C03641=1077.730,297.238,-89.064,175.217,27.521,154.780
C03642=1077.736,297.486,-89.094,175.220,27.526,154.780
C03643=1077.741,297.734,-89.125,175.222,27.530,154.781
C03644=1077.748,297.982,-89.156,175.225,27.534,154.781
C03645=1077.753,298.230,-89.187,175.228,27.538,154.782
C03646=1077.759,298.478,-89.218,175.231,27.542,154.783
C03647=1077.764,298.725,-89.249,175.234,27.547,154.783
C03648=1077.771,298.974,-89.280,175.236,27.551,154.784
C03649=1077.776,299.221,-89.312,175.240,27.555,154.785
C03650=1077.782,299.469,-89.342,175.242,27.559,154.785
C03651=1077.788,299.718,-89.373,175.245,27.563,154.786
C03652=1077.794,299.965,-89.404,175.248,27.567,154.787
C03653=1077.799,300.213,-89.435,175.251,27.571,154.787
C03654=1077.805,300.462,-89.467,175.254,27.576,154.788
C03655=1077.811,300.709,-89.498,175.257,27.580,154.789
C03656=1077.816,300.957,-89.529,175.259,27.584,154.789
C03657=1077.823,301.205,-89.561,175.262,27.588,154.790
C03658=1077.828,301.453,-89.592,175.265,27.592,154.791
C03659=1077.834,301.701,-89.624,175.268,27.596,154.791
C03660=1077.840,301.949,-89.654,175.271,27.601,154.792
C03661=1077.845,302.197,-89.686,175.273,27.605,154.793
C03662=1077.851,302.445,-89.717,175.277,27.609,154.793
C03663=1077.857,302.693,-89.748,175.280,27.614,154.794
C03664=1077.863,302.916,-89.777,175.282,27.617,154.794
C03665=1077.867,303.139,-89.805,175.284,27.621,154.795
C03666=1077.873,303.363,-89.833,175.288,27.625,154.796
C03667=1077.878,303.586,-89.862,175.290,27.629,154.796
C03668=1077.883,303.809,-89.890,175.292,27.632,154.797
C03669=1077.888,304.032,-89.919,175.295,27.636,154.797
C03670=1077.894,304.256,-89.946,175.298,27.640,154.798
C03671=1077.899,304.479,-89.975,175.300,27.644,154.799
C03672=1077.905,304.716,-90.005,175.303,27.647,154.799
C03673=1077.911,304.953,-90.034,175.306,27.651,154.800
C03674=1077.916,305.190,-90.065,175.309,27.656,154.800
C03675=1077.922,305.426,-90.096,175.311,27.660,154.801
C03676=1077.927,305.663,-90.125,175.314,27.664,154.802
C03677=1077.932,305.900,-90.155,175.317,27.667,154.802
C03678=1077.938,306.136,-90.185,175.320,27.672,154.803
C03679=1077.944,306.374,-90.216,175.322,27.676,154.804
C03680=1077.950,306.621,-90.247,175.326,27.680,154.804
C03681=1077.956,306.870,-90.279,175.329,27.684,154.805
C03682=1077.961,307.117,-90.310,175.331,27.689,154.806
C03683=1077.967,307.365,-90.342,175.334,27.693,154.806
C03684=1077.974,307.613,-90.373,175.337,27.697,154.807
C03685=1077.980,307.861,-90.405,175.340,27.701,154.808
C03686=1077.986,308.109,-90.438,175.343,27.705,154.808
C03687=1077.992,308.356,-90.469,175.346,27.709,154.809
C03688=1077.998,308.604,-90.501,175.349,27.714,154.810
C03689=1078.003,308.852,-90.532,175.352,27.718,154.810
C03690=1078.009,309.100,-90.564,175.355,27.722,154.811
C03691=1078.016,309.348,-90.596,175.358,27.727,154.812
C03692=1078.021,309.596,-90.627,175.360,27.731,154.812
C03693=1078.027,309.844,-90.659,175.364,27.735,154.813
C03694=1078.033,310.092,-90.691,175.367,27.739,154.814
C03695=1078.039,310.339,-90.722,175.370,27.743,154.814
C03696=1078.046,310.587,-90.755,175.372,27.748,154.815
C03697=1078.052,310.835,-90.787,175.376,27.752,154.816
C03698=1078.058,311.083,-90.819,175.379,27.756,154.816
C03699=1078.063,311.331,-90.851,175.381,27.760,154.817
C03700=1078.070,311.579,-90.882,175.384,27.764,154.818
C03701=1078.076,311.827,-90.914,175.387,27.769,154.818
C03702=1078.082,312.074,-90.947,175.391,27.773,154.819
C03703=1078.087,312.322,-90.979,175.393,27.777,154.820
C03704=1078.093,312.570,-91.011,175.396,27.782,154.820
C03705=1078.100,312.818,-91.042,175.399,27.786,154.821
C03706=1078.106,313.066,-91.075,175.403,27.791,154.822
C03707=1078.112,313.313,-91.107,175.405,27.794,154.822
C03708=1078.118,313.561,-91.139,175.408,27.799,154.823
C03709=1078.124,313.810,-91.171,175.411,27.803,154.824
C03710=1078.130,314.057,-91.203,175.415,27.808,154.824
C03711=1078.137,314.305,-91.235,175.417,27.812,154.825
C03712=1078.143,314.553,-91.267,175.420,27.816,154.826
C03713=1078.148,314.800,-91.299,175.423,27.820,154.826
C03714=1078.154,315.049,-91.332,175.427,27.825,154.827
C03715=1078.160,315.296,-91.365,175.429,27.829,154.828
C03716=1078.166,315.545,-91.397,175.432,27.833,154.829
C03717=1078.172,315.791,-91.429,175.435,27.838,154.829
C03718=1078.177,316.040,-91.462,175.438,27.842,154.830
C03719=1078.183,316.288,-91.494,175.441,27.847,154.831
C03720=1078.188,316.501,-91.522,175.444,27.851,154.831
C03721=1078.193,316.716,-91.550,175.446,27.855,154.832
C03722=1078.198,316.929,-91.578,175.449,27.858,154.833
C03723=1078.202,317.143,-91.606,175.451,27.862,154.833
C03724=1078.208,317.356,-91.634,175.454,27.866,154.834
C03725=1078.212,317.570,-91.662,175.456,27.870,154.835
C03726=1078.218,317.784,-91.690,175.459,27.874,154.835
C03727=1078.223,317.998,-91.718,175.461,27.878,154.836
C03728=1078.229,318.245,-91.751,175.464,27.882,154.836
C03729=1078.235,318.493,-91.784,175.468,27.887,154.837
C03730=1078.240,318.742,-91.816,175.471,27.892,154.838
C03731=1078.247,318.989,-91.849,175.474,27.896,154.839
C03732=1078.253,319.237,-91.882,175.476,27.900,154.839
C03733=1078.258,319.485,-91.914,175.479,27.905,154.840
C03734=1078.264,319.732,-91.947,175.483,27.909,154.841
C03735=1078.270,319.980,-91.980,175.486,27.914,154.842
C03736=1078.276,320.228,-92.013,175.489,27.919,154.842
C03737=1078.282,320.476,-92.045,175.491,27.923,154.843
C03738=1078.288,320.723,-92.078,175.494,27.927,154.844
C03739=1078.294,320.971,-92.111,175.498,27.932,154.845
C03740=1078.300,321.219,-92.144,175.501,27.936,154.845
C03741=1078.305,321.467,-92.177,175.504,27.941,154.846
C03742=1078.311,321.715,-92.209,175.506,27.945,154.847
C03743=1078.318,321.963,-92.242,175.509,27.950,154.848
C03744=1078.323,322.210,-92.275,175.513,27.954,154.848
C03745=1078.329,322.457,-92.308,175.516,27.959,154.849
C03746=1078.335,322.705,-92.340,175.519,27.964,154.850
C03747=1078.341,322.953,-92.374,175.522,27.968,154.851
C03748=1078.347,323.201,-92.406,175.525,27.972,154.851
C03749=1078.353,323.448,-92.440,175.528,27.977,154.852
C03750=1078.359,323.696,-92.472,175.531,27.982,154.853
C03751=1078.364,323.944,-92.506,175.534,27.987,154.854
C03752=1078.371,324.192,-92.539,175.537,27.991,154.854
C03753=1078.378,324.440,-92.572,175.541,27.995,154.855
C03754=1078.383,324.688,-92.605,175.544,28.000,154.856
C03755=1078.390,324.935,-92.638,175.546,28.005,154.857
C03756=1078.395,325.183,-92.671,175.549,28.009,154.857
C03757=1078.401,325.431,-92.704,175.552,28.014,154.858
C03758=1078.407,325.679,-92.737,175.556,28.018,154.859
C03759=1078.413,325.926,-92.770,175.559,28.023,154.859
C03760=1078.419,326.174,-92.803,175.562,28.028,154.860
C03761=1078.425,326.422,-92.836,175.565,28.032,154.861
C03762=1078.431,326.669,-92.870,175.568,28.037,154.862
C03763=1078.437,326.917,-92.903,175.571,28.041,154.863
C03764=1078.443,327.165,-92.936,175.574,28.046,154.863
C03765=1078.450,327.413,-92.969,175.577,28.050,154.864
C03766=1078.455,327.661,-93.003,175.580,28.055,154.865
C03767=1078.462,327.908,-93.036,175.584,28.060,154.866
C03768=1078.467,328.156,-93.069,175.587,28.064,154.866
C03769=1078.474,328.403,-93.102,175.590,28.069,154.867
C03770=1078.480,328.652,-93.136,175.593,28.074,154.868
C03771=1078.486,328.899,-93.169,175.596,28.078,154.869
C03772=1078.492,329.147,-93.203,175.599,28.083,154.869
C03773=1078.498,329.394,-93.235,175.602,28.088,154.870
C03774=1078.504,329.642,-93.269,175.605,28.092,154.871
C03775=1078.511,329.890,-93.303,175.608,28.097,154.872
C03776=1078.516,330.100,-93.331,175.612,28.101,154.872
C03777=1078.522,330.311,-93.360,175.614,28.105,154.873
C03778=1078.526,330.521,-93.388,175.616,28.108,154.874
C03779=1078.531,330.732,-93.416,175.620,28.113,154.874
C03780=1078.537,330.943,-93.445,175.622,28.117,154.875
C03781=1078.541,331.153,-93.473,175.624,28.120,154.876
C03782=1078.547,331.364,-93.502,175.628,28.125,154.876
C03783=1078.552,331.574,-93.531,175.630,28.129,154.877
C03784=1078.559,331.821,-93.564,175.633,28.134,154.878
C03785=1078.564,332.069,-93.597,175.636,28.138,154.879
C03786=1078.571,332.317,-93.632,175.639,28.143,154.879
C03787=1078.576,332.565,-93.665,175.643,28.148,154.880
C03788=1078.582,332.812,-93.699,175.646,28.153,154.881
C03789=1078.588,333.059,-93.733,175.649,28.158,154.882
C03790=1078.594,333.308,-93.767,175.651,28.162,154.883
C03791=1078.600,333.555,-93.801,175.654,28.167,154.884
C03792=1078.606,333.803,-93.834,175.658,28.172,154.884
C03793=1078.612,334.050,-93.868,175.661,28.177,154.885
C03794=1078.619,334.298,-93.902,175.664,28.182,154.886
C03795=1078.625,334.546,-93.936,175.667,28.186,154.887
C03796=1078.630,334.793,-93.970,175.670,28.191,154.888
C03797=1078.637,335.041,-94.004,175.674,28.196,154.888
C03798=1078.642,335.289,-94.038,175.677,28.201,154.889
C03799=1078.648,335.536,-94.072,175.680,28.206,154.890
C03800=1078.654,335.785,-94.106,175.683,28.211,154.891
C03801=1078.660,336.032,-94.140,175.686,28.216,154.892
C03802=1078.666,336.279,-94.174,175.689,28.221,154.893
C03803=1078.673,336.527,-94.208,175.693,28.225,154.893
C03804=1078.678,336.774,-94.242,175.696,28.230,154.894
C03805=1078.685,337.021,-94.276,175.699,28.235,154.895
C03806=1078.691,337.270,-94.310,175.702,28.240,154.896
C03807=1078.697,337.517,-94.344,175.705,28.245,154.897
C03808=1078.704,337.765,-94.378,175.709,28.250,154.897
C03809=1078.709,338.013,-94.412,175.712,28.255,154.898
C03810=1078.715,338.260,-94.447,175.715,28.260,154.899
C03811=1078.721,338.508,-94.481,175.718,28.265,154.900
C03812=1078.727,338.755,-94.515,175.721,28.270,154.901
C03813=1078.733,339.003,-94.550,175.725,28.275,154.902
C03814=1078.739,339.251,-94.584,175.728,28.280,154.903
C03815=1078.745,339.498,-94.618,175.731,28.285,154.904
C03816=1078.752,339.745,-94.653,175.734,28.290,154.904
C03817=1078.757,339.993,-94.687,175.737,28.295,154.905
C03818=1078.763,340.241,-94.722,175.740,28.300,154.906
C03819=1078.769,340.488,-94.756,175.744,28.305,154.907
C03820=1078.776,340.736,-94.790,175.747,28.310,154.908
C03821=1078.782,340.983,-94.824,175.750,28.315,154.909
C03822=1078.788,341.231,-94.859,175.753,28.320,154.910
C03823=1078.793,341.478,-94.894,175.757,28.326,154.910
C03824=1078.799,341.726,-94.928,175.760,28.330,154.911
C03825=1078.806,341.974,-94.963,175.764,28.335,154.912
C03826=1078.812,342.222,-94.997,175.767,28.341,154.913
C03827=1078.818,342.468,-95.032,175.770,28.346,154.914
C03828=1078.824,342.717,-95.067,175.773,28.351,154.915
C03829=1078.830,342.964,-95.101,175.776,28.356,154.916
C03830=1078.837,343.211,-95.136,175.780,28.361,154.917
C03831=1078.843,343.459,-95.170,175.783,28.366,154.917
C03832=1078.853,343.875,-95.229,175.788,28.374,154.919
C03833=1078.863,344.290,-95.287,175.794,28.383,154.920
C03834=1078.873,344.706,-95.345,175.800,28.392,154.922
C03835=1078.883,345.122,-95.404,175.804,28.400,154.923
C03836=1078.890,345.369,-95.439,175.808,28.406,154.924
C03837=1078.895,345.617,-95.474,175.811,28.411,154.925
C03838=1078.902,345.863,-95.508,175.815,28.416,154.926
C03839=1078.907,346.112,-95.543,175.818,28.422,154.927
C03840=1078.914,346.359,-95.578,175.821,28.427,154.928
C03841=1078.920,346.606,-95.613,175.824,28.432,154.929
C03842=1078.926,346.854,-95.648,175.827,28.437,154.930
C03843=1078.932,347.101,-95.683,175.830,28.442,154.931
C03844=1078.938,347.349,-95.718,175.834,28.448,154.932
C03845=1078.945,347.596,-95.753,175.838,28.453,154.933
C03846=1078.950,347.843,-95.789,175.841,28.458,154.934
C03847=1078.956,348.091,-95.823,175.844,28.463,154.934
C03848=1078.962,348.339,-95.859,175.847,28.469,154.935
C03849=1078.969,348.586,-95.893,175.850,28.474,154.936
C03850=1078.975,348.833,-95.929,175.854,28.479,154.937
C03851=1078.981,349.081,-95.964,175.857,28.485,154.938
C03852=1078.987,349.328,-95.999,175.861,28.490,154.939
C03853=1078.993,349.576,-96.035,175.864,28.496,154.940
C03854=1078.999,349.823,-96.070,175.867,28.501,154.941
C03855=1079.005,350.070,-96.105,175.870,28.506,154.942
C03856=1079.012,350.318,-96.140,175.874,28.512,154.943
C03857=1079.017,350.566,-96.175,175.877,28.517,154.944
C03858=1079.024,350.813,-96.210,175.880,28.522,154.945
C03859=1079.029,351.060,-96.246,175.884,28.528,154.946
C03860=1079.036,351.308,-96.282,175.887,28.533,154.947
C03861=1079.042,351.555,-96.317,175.890,28.538,154.948
C03862=1079.048,351.803,-96.352,175.893,28.544,154.949
C03863=1079.054,352.050,-96.388,175.897,28.549,154.950
C03864=1079.061,352.297,-96.423,175.901,28.555,154.951
C03865=1079.067,352.545,-96.459,175.904,28.560,154.952
C03866=1079.073,352.793,-96.494,175.907,28.566,154.953
C03867=1079.079,353.039,-96.529,175.910,28.571,154.954
C03868=1079.085,353.287,-96.565,175.913,28.577,154.955
C03869=1079.091,353.534,-96.601,175.917,28.583,154.956
C03870=1079.097,353.782,-96.637,175.921,28.588,154.956
C03871=1079.104,354.029,-96.672,175.924,28.593,154.957
C03872=1079.109,354.276,-96.708,175.927,28.599,154.959
C03873=1079.115,354.524,-96.743,175.930,28.605,154.960
C03874=1079.121,354.772,-96.779,175.934,28.610,154.960
C03875=1079.128,355.019,-96.815,175.937,28.616,154.961
C03876=1079.134,355.266,-96.851,175.941,28.621,154.962
C03877=1079.141,355.514,-96.886,175.944,28.627,154.964
C03878=1079.146,355.761,-96.922,175.947,28.632,154.965
C03879=1079.152,356.008,-96.958,175.951,28.638,154.966
C03880=1079.158,356.255,-96.994,175.954,28.643,154.966
C03881=1079.164,356.503,-97.030,175.957,28.649,154.968
C03882=1079.171,356.750,-97.066,175.960,28.655,154.969
C03883=1079.177,356.997,-97.101,175.965,28.660,154.970
C03884=1079.182,357.207,-97.132,175.967,28.665,154.970
C03885=1079.188,357.417,-97.162,175.970,28.670,154.971
C03886=1079.193,357.626,-97.192,175.972,28.675,154.972
C03887=1079.198,357.835,-97.223,175.976,28.679,154.973
C03888=1079.204,358.045,-97.254,175.979,28.684,154.974
C03889=1079.208,358.254,-97.284,175.981,28.689,154.975
C03890=1079.214,358.463,-97.314,175.984,28.694,154.976
C03891=1079.219,358.673,-97.345,175.988,28.699,154.977
C03892=1079.226,358.920,-97.381,175.991,28.705,154.978
C03893=1079.232,359.168,-97.417,175.994,28.710,154.979
C03894=1079.238,359.415,-97.454,175.997,28.716,154.980
C03895=1079.244,359.662,-97.489,176.001,28.722,154.981
C03896=1079.250,359.909,-97.526,176.004,28.728,154.982
C03897=1079.257,360.156,-97.562,176.008,28.733,154.983
C03898=1079.263,360.404,-97.598,176.012,28.739,154.984
C03899=1079.269,360.651,-97.634,176.015,28.745,154.985
C03900=1079.276,360.898,-97.671,176.018,28.751,154.986
C03901=1079.282,361.145,-97.707,176.021,28.757,154.987
C03902=1079.288,361.393,-97.743,176.025,28.762,154.988
C03903=1079.293,361.640,-97.780,176.028,28.769,154.989
C03904=1079.300,361.887,-97.816,176.031,28.774,154.990
C03905=1079.306,362.134,-97.853,176.036,28.780,154.991
C03906=1079.312,362.382,-97.889,176.039,28.786,154.992
C03907=1079.319,362.629,-97.925,176.042,28.792,154.993
C03908=1079.325,362.876,-97.962,176.046,28.798,154.995
C03909=1079.331,363.123,-97.998,176.049,28.804,154.996
C03910=1079.338,363.370,-98.034,176.052,28.810,154.997
C03911=1079.343,363.618,-98.071,176.056,28.816,154.998
C03912=1079.349,363.865,-98.108,176.059,28.822,154.999
C03913=1079.356,364.112,-98.144,176.063,28.827,155.000
C03914=1079.362,364.359,-98.181,176.067,28.834,155.001
C03915=1079.369,364.607,-98.218,176.070,28.839,155.002
C03916=1079.375,364.854,-98.255,176.073,28.845,155.003
C03917=1079.381,365.101,-98.291,176.077,28.852,155.005
C03918=1079.387,365.348,-98.328,176.080,28.857,155.006
C03919=1079.394,365.595,-98.364,176.083,28.863,155.007
C03920=1079.399,365.842,-98.401,176.087,28.870,155.008
C03921=1079.406,366.090,-98.437,176.091,28.876,155.009
C03922=1079.411,366.337,-98.475,176.095,28.882,155.010
C03923=1079.418,366.585,-98.511,176.098,28.888,155.011
C03924=1079.425,366.831,-98.549,176.101,28.894,155.012
C03925=1079.430,367.078,-98.586,176.105,28.900,155.014
C03926=1079.437,367.325,-98.622,176.108,28.906,155.015
C03927=1079.442,367.573,-98.659,176.111,28.912,155.016
C03928=1079.449,367.819,-98.696,176.115,28.918,155.017
C03929=1079.456,368.067,-98.733,176.119,28.925,155.018
C03930=1079.462,368.314,-98.770,176.123,28.931,155.019
C03931=1079.468,368.561,-98.806,176.126,28.937,155.021
C03932=1079.474,368.808,-98.844,176.129,28.944,155.022
C03933=1079.480,369.055,-98.881,176.133,28.950,155.023
C03934=1079.487,369.303,-98.919,176.136,28.956,155.024
C03935=1079.493,369.550,-98.955,176.140,28.962,155.025
C03936=1079.499,369.797,-98.992,176.143,28.968,155.026
C03937=1079.505,370.044,-99.029,176.146,28.974,155.028
C03938=1079.512,370.291,-99.066,176.150,28.981,155.029
C03939=1079.518,370.538,-99.104,176.154,28.987,155.030
C03940=1079.524,370.755,-99.137,176.157,28.993,155.031
C03941=1079.529,370.973,-99.169,176.160,28.998,155.032
C03942=1079.535,371.190,-99.202,176.163,29.004,155.033
C03943=1079.541,371.408,-99.235,176.166,29.009,155.034
C03944=1079.546,371.626,-99.268,176.170,29.015,155.035
C03945=1079.552,371.843,-99.300,176.173,29.021,155.036
C03946=1079.557,372.060,-99.333,176.176,29.026,155.037
C03947=1079.563,372.278,-99.367,176.179,29.032,155.038
C03948=1079.569,372.525,-99.404,176.182,29.038,155.040
C03949=1079.576,372.772,-99.441,176.187,29.045,155.041
C03950=1079.582,373.019,-99.479,176.190,29.051,155.042
C03951=1079.588,373.267,-99.516,176.194,29.057,155.043
C03952=1079.595,373.514,-99.554,176.197,29.064,155.044
C03953=1079.601,373.761,-99.591,176.201,29.070,155.046
C03954=1079.608,374.007,-99.628,176.204,29.077,155.047
C03955=1079.614,374.255,-99.666,176.208,29.084,155.048
C03956=1079.620,374.502,-99.704,176.211,29.090,155.049
C03957=1079.626,374.749,-99.741,176.214,29.096,155.051
C03958=1079.632,374.996,-99.779,176.218,29.103,155.052
C03959=1079.639,375.242,-99.817,176.222,29.109,155.053
C03960=1079.645,375.489,-99.854,176.226,29.116,155.054
C03961=1079.651,375.737,-99.892,176.229,29.123,155.056
C03962=1079.657,375.983,-99.930,176.233,29.130,155.057
C03963=1079.664,376.231,-99.968,176.237,29.136,155.058
C03964=1079.670,376.477,-100.006,176.240,29.143,155.060
C03965=1079.677,376.725,-100.044,176.244,29.150,155.061
C03966=1079.683,376.971,-100.081,176.247,29.156,155.062
C03967=1079.689,377.219,-100.120,176.251,29.163,155.063
C03968=1079.695,377.466,-100.157,176.254,29.170,155.065
C03969=1079.702,377.713,-100.195,176.259,29.176,155.066
C03970=1079.708,377.959,-100.233,176.262,29.183,155.067
C03971=1079.715,378.207,-100.271,176.266,29.190,155.069
C03972=1079.721,378.453,-100.309,176.269,29.197,155.070
C03973=1079.727,378.701,-100.347,176.273,29.203,155.071
C03974=1079.733,378.947,-100.385,176.276,29.210,155.073
C03975=1079.740,379.195,-100.423,176.280,29.217,155.074
C03976=1079.746,379.441,-100.462,176.284,29.224,155.075
C03977=1079.753,379.688,-100.499,176.287,29.231,155.076
C03978=1079.759,379.935,-100.537,176.291,29.237,155.078
C03979=1079.766,380.182,-100.576,176.294,29.244,155.079
C03980=1079.773,380.429,-100.614,176.299,29.251,155.080
C03981=1079.778,380.676,-100.652,176.303,29.258,155.082
C03982=1079.785,380.923,-100.690,176.306,29.265,155.083
C03983=1079.791,381.169,-100.728,176.310,29.272,155.084
C03984=1079.798,381.416,-100.767,176.313,29.279,155.086
C03985=1079.804,381.664,-100.805,176.317,29.285,155.087
C03986=1079.811,381.911,-100.843,176.321,29.293,155.089
C03987=1079.817,382.157,-100.882,176.324,29.300,155.090
C03988=1079.824,382.405,-100.920,176.328,29.306,155.091
C03989=1079.830,382.651,-100.958,176.332,29.314,155.093
C03990=1079.837,382.897,-100.997,176.335,29.321,155.094
C03991=1079.843,383.145,-101.035,176.339,29.328,155.095
C03992=1079.849,383.391,-101.074,176.343,29.335,155.097
C03993=1079.855,383.638,-101.113,176.347,29.342,155.098
C03994=1079.862,383.886,-101.151,176.351,29.349,155.100
C03995=1079.868,384.132,-101.190,176.354,29.356,155.101
C03996=1079.874,384.364,-101.226,176.358,29.363,155.102
C03997=1079.880,384.595,-101.263,176.361,29.370,155.104
C03998=1079.886,384.827,-101.299,176.364,29.377,155.105
C03999=1079.892,385.059,-101.336,176.368,29.383,155.106
C04000=1079.898,385.291,-101.372,176.371,29.390,155.108
C04001=1079.905,385.523,-101.408,176.376,29.397,155.109
C04002=1079.910,385.755,-101.445,176.379,29.404,155.110
C04003=1079.917,385.987,-101.481,176.382,29.411,155.112
C04004=1079.923,386.234,-101.520,176.386,29.418,155.113
C04005=1079.929,386.480,-101.559,176.390,29.425,155.115
C04006=1079.936,386.727,-101.597,176.394,29.433,155.116
C04007=1079.943,386.974,-101.636,176.397,29.440,155.118
C04008=1079.949,387.221,-101.676,176.401,29.447,155.119
C04009=1079.955,387.467,-101.714,176.405,29.455,155.120
C04010=1079.962,387.714,-101.753,176.408,29.462,155.122
C04011=1079.968,387.961,-101.792,176.413,29.469,155.123
C04012=1079.974,388.208,-101.831,176.417,29.477,155.125
C04013=1079.981,388.455,-101.870,176.421,29.484,155.126
C04014=1079.988,388.701,-101.909,176.424,29.492,155.128
C04015=1079.994,388.949,-101.948,176.428,29.499,155.129
C04016=1080.001,389.194,-101.988,176.432,29.507,155.131
C04017=1080.008,389.441,-102.026,176.436,29.514,155.132
C04018=1080.014,389.688,-102.066,176.439,29.521,155.134
C04019=1080.020,389.935,-102.105,176.443,29.529,155.135
C04020=1080.027,390.182,-102.144,176.447,29.537,155.137
C04021=1080.034,390.428,-102.184,176.451,29.544,155.138
C04022=1080.040,390.675,-102.223,176.455,29.552,155.140
C04023=1080.047,390.922,-102.261,176.458,29.559,155.141
C04024=1080.054,391.168,-102.302,176.463,29.567,155.143
C04025=1080.060,391.415,-102.340,176.467,29.574,155.144
C04026=1080.066,391.662,-102.380,176.471,29.582,155.146
C04027=1080.074,391.908,-102.419,176.475,29.590,155.147
C04028=1080.080,392.156,-102.459,176.478,29.597,155.149
C04029=1080.087,392.402,-102.498,176.482,29.606,155.151
C04030=1080.093,392.649,-102.538,176.486,29.613,155.152
C04031=1080.099,392.895,-102.578,176.490,29.621,155.154
C04032=1080.106,393.142,-102.617,176.494,29.629,155.155
C04033=1080.112,393.389,-102.657,176.497,29.636,155.157
C04034=1080.119,393.636,-102.696,176.501,29.644,155.158
C04035=1080.126,393.882,-102.736,176.505,29.652,155.160
C04036=1080.132,394.129,-102.776,176.509,29.660,155.162
C04037=1080.139,394.375,-102.815,176.513,29.668,155.163
C04038=1080.145,394.622,-102.855,176.518,29.676,155.165
C04039=1080.152,394.869,-102.896,176.521,29.684,155.167
C04040=1080.159,395.116,-102.934,176.525,29.692,155.168
C04041=1080.165,395.363,-102.975,176.529,29.700,155.170
C04042=1080.172,395.609,-103.015,176.533,29.708,155.171
C04043=1080.178,395.856,-103.055,176.537,29.716,155.173
C04044=1080.185,396.102,-103.094,176.541,29.724,155.175
C04045=1080.191,396.349,-103.134,176.545,29.732,155.176
C04046=1080.198,396.596,-103.174,176.548,29.740,155.178
C04047=1080.205,396.843,-103.214,176.552,29.748,155.180
C04048=1080.211,397.089,-103.255,176.556,29.756,155.181
C04049=1080.218,397.335,-103.294,176.560,29.765,155.183
C04050=1080.225,397.582,-103.334,176.564,29.773,155.185
C04051=1080.232,397.829,-103.375,176.568,29.781,155.186
C04052=1080.238,398.068,-103.414,176.572,29.789,155.188
C04053=1080.244,398.307,-103.452,176.577,29.797,155.190
C04054=1080.250,398.546,-103.491,176.580,29.805,155.191
C04055=1080.258,398.785,-103.530,176.584,29.813,155.193
C04056=1080.264,399.024,-103.569,176.588,29.821,155.195
C04057=1080.270,399.263,-103.608,176.592,29.829,155.196
C04058=1080.276,399.502,-103.647,176.595,29.837,155.198
C04059=1080.283,399.741,-103.686,176.599,29.845,155.200
C04060=1080.289,399.988,-103.727,176.603,29.854,155.201
C04061=1080.296,400.234,-103.767,176.607,29.862,155.203
C04062=1080.303,400.481,-103.808,176.611,29.870,155.205
C04063=1080.309,400.727,-103.848,176.615,29.879,155.207
C04064=1080.316,400.974,-103.888,176.620,29.887,155.208
C04065=1080.323,401.221,-103.929,176.624,29.896,155.210
C04066=1080.329,401.467,-103.970,176.628,29.904,155.212
C04067=1080.336,401.714,-104.011,176.632,29.913,155.214
C04068=1080.342,401.961,-104.051,176.636,29.922,155.215
C04069=1080.349,402.207,-104.092,176.640,29.930,155.217
C04070=1080.356,402.454,-104.132,176.644,29.939,155.219
C04071=1080.363,402.700,-104.173,176.648,29.947,155.221
C04072=1080.370,402.947,-104.214,176.652,29.956,155.223
C04073=1080.376,403.193,-104.255,176.656,29.965,155.224
C04074=1080.383,403.440,-104.295,176.660,29.973,155.226
C04075=1080.390,403.686,-104.336,176.664,29.982,155.228
C04076=1080.397,403.933,-104.376,176.668,29.991,155.230
C04077=1080.403,404.180,-104.418,176.672,30.000,155.232
C04078=1080.410,404.426,-104.459,176.677,30.009,155.234
C04079=1080.416,404.673,-104.499,176.682,30.017,155.235
C04080=1080.424,404.919,-104.540,176.686,30.027,155.237
C04081=1080.430,405.165,-104.582,176.690,30.035,155.239
C04082=1080.437,405.413,-104.622,176.694,30.044,155.241
C04083=1080.443,405.659,-104.663,176.698,30.053,155.243
C04084=1080.451,405.905,-104.705,176.702,30.062,155.245
C04085=1080.457,406.152,-104.746,176.706,30.071,155.247
C04086=1080.464,406.398,-104.787,176.710,30.080,155.249
C04087=1080.471,406.645,-104.828,176.715,30.089,155.250
C04088=1080.477,406.891,-104.869,176.719,30.098,155.252
C04089=1080.484,407.138,-104.910,176.723,30.107,155.254
C04090=1080.491,407.385,-104.952,176.727,30.116,155.256
C04091=1080.497,407.631,-104.993,176.731,30.126,155.258
C04092=1080.504,407.878,-105.035,176.736,30.135,155.260
C04093=1080.511,408.124,-105.076,176.741,30.144,155.262
C04094=1080.517,408.370,-105.118,176.745,30.153,155.264
C04095=1080.524,408.617,-105.159,176.749,30.162,155.266
C04096=1080.530,408.863,-105.200,176.753,30.172,155.268
C04097=1080.538,409.109,-105.242,176.757,30.181,155.270
C04098=1080.544,409.356,-105.284,176.762,30.191,155.272
C04099=1080.551,409.602,-105.325,176.766,30.200,155.274
C04100=1080.558,409.849,-105.367,176.770,30.209,155.276
C04101=1080.565,410.096,-105.408,176.774,30.219,155.278
C04102=1080.572,410.342,-105.451,176.779,30.228,155.280
C04103=1080.579,410.588,-105.491,176.783,30.238,155.282
C04104=1080.585,410.835,-105.533,176.787,30.247,155.284
C04105=1080.593,411.081,-105.575,176.792,30.257,155.286
C04106=1080.599,411.328,-105.617,176.797,30.267,155.288
C04107=1080.606,411.574,-105.659,176.801,30.276,155.290
C04108=1080.612,411.814,-105.700,176.805,30.285,155.292
C04109=1080.619,412.054,-105.741,176.809,30.295,155.294
C04110=1080.626,412.294,-105.781,176.813,30.304,155.296
C04111=1080.633,412.534,-105.822,176.818,30.314,155.298
C04112=1080.640,412.774,-105.862,176.822,30.323,155.300
C04113=1080.647,413.014,-105.903,176.826,30.332,155.302
C04114=1080.653,413.255,-105.945,176.830,30.342,155.304
C04115=1080.660,413.494,-105.986,176.836,30.352,155.306
C04116=1080.667,413.741,-106.027,176.840,30.362,155.308
C04117=1080.674,413.987,-106.070,176.844,30.371,155.310
C04118=1080.681,414.234,-106.112,176.849,30.381,155.313
C04119=1080.688,414.480,-106.154,176.853,30.391,155.315
C04120=1080.695,414.727,-106.196,176.857,30.401,155.317
C04121=1080.702,414.973,-106.239,176.862,30.411,155.319
C04122=1080.709,415.219,-106.281,176.866,30.420,155.321
C04123=1080.716,415.466,-106.323,176.871,30.431,155.323
C04124=1080.723,415.712,-106.365,176.875,30.441,155.325
C04125=1080.730,415.958,-106.408,176.881,30.451,155.327
C04126=1080.737,416.205,-106.450,176.885,30.461,155.330
C04127=1080.743,416.451,-106.493,176.890,30.471,155.332
C04128=1080.751,416.697,-106.535,176.894,30.481,155.334
C04129=1080.758,416.943,-106.577,176.898,30.491,155.336
C04130=1080.765,417.189,-106.620,176.903,30.502,155.339
C04131=1080.772,417.436,-106.662,176.907,30.512,155.341
C04132=1080.778,417.682,-106.705,176.912,30.523,155.343
C04133=1080.786,417.928,-106.748,176.916,30.533,155.345
C04134=1080.792,418.174,-106.791,176.921,30.543,155.348
C04135=1080.799,418.420,-106.833,176.927,30.554,155.350
C04136=1080.806,418.666,-106.876,176.931,30.564,155.352
C04137=1080.813,418.913,-106.918,176.936,30.575,155.354
C04138=1080.820,419.158,-106.961,176.940,30.585,155.357
C04139=1080.828,419.405,-107.004,176.945,30.595,155.359
C04140=1080.834,419.652,-107.047,176.949,30.606,155.361
C04141=1080.842,419.897,-107.090,176.954,30.617,155.364
C04142=1080.849,420.144,-107.133,176.958,30.627,155.366
C04143=1080.856,420.389,-107.176,176.964,30.638,155.368
C04144=1080.863,420.636,-107.219,176.969,30.649,155.371
C04145=1080.870,420.882,-107.262,176.973,30.659,155.373
C04146=1080.877,421.128,-107.305,176.978,30.670,155.375
C04147=1080.884,421.374,-107.348,176.983,30.681,155.378
C04148=1080.891,421.621,-107.391,176.987,30.692,155.380
C04149=1080.898,421.867,-107.435,176.992,30.702,155.382
C04150=1080.905,422.113,-107.478,176.997,30.713,155.385
C04151=1080.913,422.360,-107.521,177.002,30.724,155.387
C04152=1080.920,422.605,-107.564,177.007,30.735,155.390
C04153=1080.926,422.851,-107.608,177.012,30.746,155.392
C04154=1080.934,423.097,-107.651,177.016,30.757,155.394
C04155=1080.941,423.344,-107.694,177.021,30.768,155.397
C04156=1080.947,423.590,-107.738,177.026,30.780,155.399
C04157=1080.955,423.835,-107.781,177.030,30.791,155.402
C04158=1080.962,424.082,-107.825,177.036,30.802,155.404
C04159=1080.969,424.328,-107.869,177.041,30.814,155.407
C04160=1080.976,424.573,-107.912,177.046,30.825,155.409
C04161=1080.984,424.820,-107.956,177.050,30.836,155.412
C04162=1080.990,425.066,-107.999,177.055,30.847,155.414
C04163=1080.998,425.312,-108.043,177.060,30.859,155.417
C04164=1081.005,425.563,-108.087,177.066,30.870,155.419
C04165=1081.013,425.813,-108.132,177.071,30.882,155.422
C04166=1081.020,426.064,-108.177,177.076,30.894,155.425
C04167=1081.027,426.314,-108.222,177.081,30.905,155.427
C04168=1081.035,426.560,-108.265,177.085,30.917,155.430
C04169=1081.041,426.806,-108.309,177.090,30.928,155.432
C04170=1081.049,427.053,-108.353,177.096,30.940,155.435
C04171=1081.056,427.298,-108.397,177.101,30.952,155.438
C04172=1081.063,427.544,-108.441,177.106,30.963,155.440
C04173=1081.071,427.791,-108.484,177.111,30.975,155.443
C04174=1081.078,428.036,-108.529,177.116,30.987,155.445
C04175=1081.086,428.283,-108.573,177.121,30.998,155.448
C04176=1081.092,428.528,-108.617,177.126,31.010,155.451
C04177=1081.100,428.774,-108.661,177.131,31.022,155.453
C04178=1081.108,429.020,-108.706,177.136,31.034,155.456
C04179=1081.114,429.266,-108.750,177.141,31.046,155.459
C04180=1081.122,429.512,-108.794,177.147,31.058,155.461
C04181=1081.129,429.757,-108.838,177.152,31.070,155.464
C04182=1081.136,430.004,-108.883,177.157,31.082,155.467
C04183=1081.144,430.250,-108.927,177.162,31.094,155.470
C04184=1081.151,430.495,-108.972,177.167,31.106,155.472
C04185=1081.158,430.741,-109.017,177.173,31.118,155.475
C04186=1081.166,430.987,-109.061,177.178,31.131,155.478
C04187=1081.173,431.234,-109.105,177.183,31.143,155.481
C04188=1081.180,431.479,-109.150,177.188,31.155,155.483
C04189=1081.188,431.725,-109.194,177.194,31.167,155.486
C04190=1081.195,431.971,-109.239,177.199,31.180,155.489
C04191=1081.202,432.217,-109.284,177.204,31.192,155.492
C04192=1081.210,432.462,-109.328,177.209,31.205,155.494
C04193=1081.217,432.708,-109.373,177.215,31.217,155.497
C04194=1081.225,432.954,-109.418,177.220,31.230,155.500
C04195=1081.232,433.199,-109.463,177.225,31.243,155.503
C04196=1081.239,433.445,-109.508,177.230,31.255,155.506
C04197=1081.246,433.691,-109.553,177.237,31.268,155.509
C04198=1081.254,433.937,-109.598,177.242,31.281,155.512
C04199=1081.261,434.182,-109.643,177.247,31.293,155.515
C04200=1081.269,434.428,-109.688,177.252,31.306,155.518
C04201=1081.276,434.674,-109.733,177.258,31.319,155.520
C04202=1081.284,434.920,-109.779,177.263,31.332,155.523
C04203=1081.291,435.166,-109.824,177.268,31.345,155.526
C04204=1081.298,435.411,-109.869,177.275,31.358,155.529
C04205=1081.305,435.657,-109.914,177.280,31.371,155.532
C04206=1081.313,435.902,-109.960,177.285,31.384,155.535
C04207=1081.320,436.148,-110.005,177.290,31.397,155.538
C04208=1081.328,436.394,-110.050,177.296,31.410,155.541
C04209=1081.336,436.639,-110.096,177.302,31.424,155.544
C04210=1081.343,436.885,-110.141,177.307,31.437,155.547
C04211=1081.351,437.131,-110.187,177.313,31.450,155.550
C04212=1081.358,437.376,-110.232,177.318,31.463,155.554
C04213=1081.366,437.621,-110.278,177.324,31.477,155.557
C04214=1081.374,437.868,-110.323,177.330,31.490,155.560
C04215=1081.381,438.114,-110.369,177.335,31.503,155.563
C04216=1081.389,438.359,-110.414,177.341,31.517,155.566
C04217=1081.397,438.604,-110.460,177.347,31.531,155.569
C04218=1081.404,438.850,-110.506,177.352,31.544,155.572
C04219=1081.412,439.095,-110.551,177.358,31.558,155.575
C04220=1081.419,439.347,-110.598,177.364,31.572,155.579
C04221=1081.428,439.599,-110.645,177.370,31.586,155.582
C04222=1081.435,439.850,-110.693,177.376,31.600,155.585
C04223=1081.443,440.102,-110.740,177.382,31.614,155.588
C04224=1081.451,440.347,-110.786,177.387,31.628,155.592
C04225=1081.458,440.592,-110.831,177.394,31.642,155.595
C04226=1081.467,440.838,-110.878,177.399,31.656,155.598
C04227=1081.474,441.084,-110.924,177.405,31.670,155.601
C04228=1081.481,441.329,-110.970,177.411,31.685,155.605
C04229=1081.489,441.574,-111.016,177.416,31.698,155.608
C04230=1081.497,441.820,-111.063,177.423,31.713,155.611
C04231=1081.505,442.065,-111.109,177.428,31.727,155.615
C04232=1081.512,442.311,-111.155,177.435,31.741,155.618
C04233=1081.520,442.557,-111.202,177.440,31.755,155.621
C04234=1081.528,442.802,-111.248,177.447,31.770,155.625
C04235=1081.536,443.048,-111.295,177.452,31.785,155.628
C04236=1081.544,443.293,-111.341,177.458,31.799,155.631
C04237=1081.550,443.538,-111.388,177.464,31.814,155.635
C04238=1081.559,443.784,-111.434,177.470,31.828,155.638
C04239=1081.566,444.029,-111.481,177.477,31.843,155.642
C04240=1081.575,444.274,-111.528,177.482,31.857,155.645
C04241=1081.582,444.520,-111.575,177.489,31.872,155.649
C04242=1081.590,444.765,-111.622,177.494,31.887,155.652
C04243=1081.597,445.011,-111.668,177.501,31.902,155.656
C04244=1081.606,445.256,-111.715,177.507,31.917,155.659
C04245=1081.613,445.501,-111.762,177.513,31.932,155.663
C04246=1081.621,445.747,-111.810,177.520,31.947,155.666
C04247=1081.629,445.991,-111.856,177.525,31.962,155.670
C04248=1081.637,446.237,-111.903,177.531,31.977,155.673
C04249=1081.645,446.482,-111.950,177.536,31.992,155.677
C04250=1081.653,446.728,-111.997,177.542,32.007,155.681
C04251=1081.661,446.974,-112.044,177.546,32.022,155.684
C04252=1081.668,447.218,-112.092,177.551,32.037,155.688
C04253=1081.677,447.464,-112.139,177.556,32.052,155.691
C04254=1081.684,447.710,-112.186,177.560,32.067,155.695
C04255=1081.692,447.954,-112.234,177.564,32.082,155.699
C04256=1081.700,448.200,-112.281,177.568,32.097,155.702
C04257=1081.709,448.445,-112.329,177.571,32.112,155.706
C04258=1081.716,448.691,-112.376,177.575,32.127,155.710
C04259=1081.724,448.935,-112.424,177.578,32.141,155.714
C04260=1081.732,449.179,-112.471,177.581,32.157,155.717
C04261=1081.741,449.425,-112.517,177.584,32.171,155.721
C04262=1081.753,449.671,-112.563,177.587,32.184,155.724
C04263=1081.765,449.916,-112.608,177.590,32.197,155.727
C04264=1081.398,449.910,-112.826,177.562,32.369,155.773
C04265=1081.385,449.664,-112.781,177.558,32.356,155.770
C04266=1081.374,449.419,-112.736,177.555,32.342,155.767
C04267=1081.364,449.174,-112.688,177.553,32.328,155.763
C04268=1081.356,448.929,-112.641,177.550,32.314,155.759
C04269=1081.345,448.584,-112.574,177.545,32.292,155.754
C04270=1081.333,448.239,-112.508,177.539,32.271,155.749
C04271=1081.322,447.893,-112.440,177.534,32.251,155.744
C04272=1081.311,447.549,-112.374,177.528,32.229,155.739
C04273=1081.303,447.303,-112.327,177.523,32.214,155.735
C04274=1081.295,447.058,-112.280,177.519,32.199,155.731
C04275=1081.287,446.813,-112.232,177.514,32.184,155.728
C04276=1081.279,446.568,-112.185,177.508,32.169,155.724
C04277=1081.271,446.322,-112.138,177.502,32.154,155.720
C04278=1081.263,446.078,-112.090,177.497,32.139,155.717
C04279=1081.256,445.832,-112.043,177.491,32.124,155.713
C04280=1081.247,445.586,-111.996,177.484,32.109,155.710
C04281=1081.240,445.341,-111.949,177.479,32.094,155.706
C04282=1081.232,445.095,-111.902,177.472,32.079,155.703
C04283=1081.224,444.850,-111.856,177.466,32.064,155.699
C04284=1081.216,444.605,-111.808,177.460,32.049,155.696
C04285=1081.208,444.360,-111.762,177.453,32.034,155.692
C04286=1081.200,444.114,-111.715,177.448,32.020,155.689
C04287=1081.193,443.869,-111.668,177.441,32.005,155.685
C04288=1081.185,443.623,-111.621,177.435,31.991,155.682
C04289=1081.177,443.379,-111.575,177.429,31.976,155.678
C04290=1081.169,443.132,-111.528,177.422,31.961,155.675
C04291=1081.161,442.887,-111.482,177.417,31.947,155.671
C04292=1081.153,442.643,-111.435,177.410,31.933,155.668
C04293=1081.146,442.397,-111.388,177.405,31.918,155.665
C04294=1081.138,442.151,-111.342,177.398,31.904,155.661
C04295=1081.130,441.905,-111.295,177.393,31.889,155.658
C04296=1081.122,441.660,-111.249,177.386,31.875,155.655
C04297=1081.115,441.415,-111.203,177.381,31.861,155.651
C04298=1081.107,441.169,-111.156,177.374,31.847,155.648
C04299=1081.099,440.924,-111.110,177.369,31.833,155.645
C04300=1081.091,440.679,-111.064,177.362,31.819,155.641
C04301=1081.080,440.297,-110.992,177.354,31.797,155.636
C04302=1081.068,439.915,-110.921,177.345,31.775,155.631
C04303=1081.056,439.535,-110.849,177.336,31.754,155.626
C04304=1081.044,439.153,-110.778,177.326,31.733,155.621
C04305=1081.037,438.908,-110.733,177.320,31.719,155.618
C04306=1081.029,438.662,-110.687,177.315,31.705,155.615
C04307=1081.021,438.416,-110.641,177.309,31.692,155.612
C04308=1081.013,438.171,-110.595,177.304,31.678,155.609
C04309=1081.005,437.925,-110.550,177.297,31.665,155.606
C04310=1080.998,437.680,-110.504,177.292,31.652,155.603
C04311=1080.990,437.434,-110.458,177.286,31.638,155.600
C04312=1080.983,437.189,-110.413,177.280,31.625,155.597
C04313=1080.975,436.943,-110.367,177.274,31.611,155.593
C04314=1080.967,436.698,-110.321,177.269,31.598,155.590
C04315=1080.960,436.452,-110.276,177.264,31.585,155.587
C04316=1080.952,436.206,-110.231,177.257,31.572,155.584
C04317=1080.944,435.960,-110.185,177.252,31.558,155.581
C04318=1080.937,435.714,-110.140,177.246,31.546,155.578
C04319=1080.930,435.470,-110.095,177.241,31.533,155.575
C04320=1080.922,435.224,-110.050,177.236,31.519,155.572
C04321=1080.915,434.978,-110.004,177.230,31.507,155.569
C04322=1080.907,434.732,-109.959,177.224,31.494,155.566
C04323=1080.900,434.487,-109.913,177.219,31.481,155.563
C04324=1080.892,434.241,-109.869,177.213,31.468,155.561
C04325=1080.885,433.995,-109.823,177.208,31.455,155.558
C04326=1080.877,433.749,-109.778,177.202,31.443,155.555
C04327=1080.870,433.503,-109.733,177.197,31.430,155.552
C04328=1080.862,433.258,-109.687,177.192,31.417,155.549
C04329=1080.856,433.012,-109.643,177.186,31.404,155.546
C04330=1080.848,432.766,-109.598,177.181,31.392,155.543
C04331=1080.841,432.520,-109.553,177.175,31.379,155.540
C04332=1080.833,432.274,-109.509,177.169,31.366,155.537
C04333=1080.826,432.028,-109.464,177.164,31.354,155.535
C04334=1080.819,431.783,-109.419,177.159,31.342,155.532
C04335=1080.812,431.537,-109.374,177.154,31.329,155.529
C04336=1080.804,431.291,-109.330,177.148,31.317,155.526
C04337=1080.796,431.045,-109.285,177.143,31.305,155.523
C04338=1080.789,430.799,-109.240,177.138,31.292,155.521
C04339=1080.781,430.554,-109.196,177.132,31.280,155.518
C04340=1080.774,430.308,-109.151,177.127,31.268,155.515
C04341=1080.767,430.062,-109.106,177.122,31.256,155.512
C04342=1080.759,429.817,-109.062,177.116,31.244,155.510
C04343=1080.752,429.570,-109.018,177.111,31.232,155.507
C04344=1080.745,429.324,-108.973,177.107,31.220,155.504
C04345=1080.737,429.079,-108.929,177.101,31.208,155.502
C04346=1080.730,428.832,-108.885,177.096,31.196,155.499
C04347=1080.722,428.587,-108.841,177.091,31.184,155.496
C04348=1080.716,428.341,-108.797,177.086,31.172,155.494
C04349=1080.709,428.095,-108.752,177.080,31.160,155.491
C04350=1080.701,427.849,-108.708,177.075,31.148,155.488
C04351=1080.694,427.603,-108.664,177.070,31.137,155.486
C04352=1080.686,427.357,-108.620,177.065,31.125,155.483
C04353=1080.679,427.112,-108.576,177.060,31.114,155.480
C04354=1080.672,426.865,-108.532,177.055,31.102,155.478
C04355=1080.665,426.619,-108.488,177.050,31.091,155.475
C04356=1080.657,426.373,-108.444,177.045,31.079,155.473
C04357=1080.650,426.121,-108.399,177.039,31.067,155.470
C04358=1080.642,425.869,-108.354,177.034,31.056,155.467
C04359=1080.635,425.617,-108.310,177.029,31.044,155.465
C04360=1080.628,425.365,-108.264,177.024,31.032,155.462
C04361=1080.620,425.119,-108.221,177.019,31.021,155.460
C04362=1080.613,424.873,-108.177,177.014,31.009,155.457
C04363=1080.606,424.626,-108.133,177.009,30.998,155.455
C04364=1080.599,424.381,-108.090,177.004,30.987,155.452
C04365=1080.592,424.135,-108.046,176.999,30.976,155.450
C04366=1080.584,423.888,-108.002,176.994,30.964,155.447
C04367=1080.577,423.643,-107.959,176.989,30.953,155.445
C04368=1080.571,423.397,-107.915,176.984,30.942,155.442
C04369=1080.563,423.150,-107.872,176.980,30.931,155.440
C04370=1080.556,422.905,-107.828,176.974,30.920,155.437
C04371=1080.549,422.659,-107.786,176.969,30.909,155.435
C04372=1080.542,422.412,-107.742,176.965,30.898,155.432
C04373=1080.535,422.166,-107.698,176.960,30.887,155.430
C04374=1080.528,421.921,-107.655,176.955,30.876,155.428
C04375=1080.520,421.674,-107.612,176.950,30.865,155.425
C04376=1080.513,421.428,-107.569,176.945,30.854,155.423
C04377=1080.507,421.182,-107.525,176.940,30.843,155.421
C04378=1080.499,420.935,-107.482,176.936,30.833,155.418
C04379=1080.492,420.689,-107.439,176.931,30.822,155.416
C04380=1080.485,420.443,-107.396,176.926,30.812,155.413
C04381=1080.478,420.197,-107.353,176.921,30.800,155.411
C04382=1080.470,419.950,-107.310,176.916,30.790,155.409
C04383=1080.463,419.705,-107.267,176.912,30.779,155.406
C04384=1080.456,419.458,-107.224,176.907,30.769,155.404
C04385=1080.449,419.213,-107.181,176.902,30.758,155.402
C04386=1080.442,418.966,-107.139,176.897,30.748,155.400
C04387=1080.435,418.719,-107.096,176.893,30.737,155.397
C04388=1080.428,418.474,-107.052,176.888,30.727,155.395
C04389=1080.421,418.227,-107.010,176.884,30.716,155.393
C04390=1080.414,417.981,-106.967,176.878,30.706,155.390
C04391=1080.407,417.735,-106.925,176.874,30.696,155.388
C04392=1080.400,417.489,-106.882,176.869,30.685,155.386
C04393=1080.393,417.243,-106.839,176.865,30.675,155.384
C04394=1080.386,416.997,-106.797,176.860,30.664,155.381
C04395=1080.380,416.750,-106.754,176.856,30.655,155.379
C04396=1080.373,416.504,-106.711,176.850,30.644,155.377
C04397=1080.365,416.257,-106.669,176.846,30.634,155.375
C04398=1080.358,416.011,-106.627,176.841,30.624,155.373
C04399=1080.351,415.765,-106.584,176.837,30.614,155.370
C04400=1080.344,415.519,-106.542,176.833,30.604,155.368
C04401=1080.337,415.272,-106.499,176.828,30.594,155.366
C04402=1080.330,415.026,-106.456,176.823,30.584,155.364
C04403=1080.323,414.779,-106.415,176.818,30.573,155.362
C04404=1080.316,414.533,-106.373,176.814,30.564,155.360
C04405=1080.309,414.287,-106.330,176.809,30.554,155.358
C04406=1080.302,414.041,-106.288,176.805,30.544,155.355
C04407=1080.295,413.794,-106.246,176.801,30.534,155.353
C04408=1080.288,413.548,-106.204,176.795,30.524,155.351
C04409=1080.281,413.308,-106.163,176.791,30.515,155.349
C04410=1080.274,413.067,-106.122,176.787,30.505,155.347
C04411=1080.268,412.826,-106.081,176.783,30.496,155.345
C04412=1080.260,412.585,-106.040,176.778,30.486,155.343
C04413=1080.254,412.344,-105.999,176.774,30.476,155.341
C04414=1080.247,412.103,-105.958,176.769,30.467,155.339
C04415=1080.240,411.863,-105.917,176.765,30.458,155.337
C04416=1080.234,411.622,-105.876,176.761,30.448,155.335
C04417=1080.227,411.376,-105.835,176.756,30.439,155.333
C04418=1080.220,411.129,-105.792,176.752,30.429,155.331
C04419=1080.213,410.882,-105.750,176.748,30.420,155.329
C04420=1080.206,410.636,-105.708,176.744,30.410,155.327
C04421=1080.200,410.390,-105.667,176.738,30.400,155.325
C04422=1080.193,410.144,-105.626,176.734,30.391,155.323
C04423=1080.186,409.897,-105.583,176.730,30.382,155.321
C04424=1080.178,409.651,-105.542,176.726,30.372,155.319
C04425=1080.172,409.404,-105.500,176.721,30.363,155.317
C04426=1080.165,409.158,-105.459,176.717,30.354,155.315
C04427=1080.158,408.912,-105.417,176.713,30.344,155.313
C04428=1080.152,408.665,-105.375,176.708,30.335,155.311
C04429=1080.145,408.419,-105.334,176.704,30.326,155.309
C04430=1080.139,408.172,-105.292,176.699,30.316,155.307
C04431=1080.131,407.925,-105.251,176.695,30.307,155.305
C04432=1080.125,407.679,-105.210,176.691,30.298,155.303
C04433=1080.118,407.433,-105.168,176.687,30.289,155.301
C04434=1080.112,407.186,-105.126,176.683,30.280,155.299
C04435=1080.105,406.940,-105.086,176.679,30.271,155.297
C04436=1080.098,406.693,-105.044,176.674,30.262,155.295
C04437=1080.092,406.447,-105.003,176.669,30.252,155.293
C04438=1080.084,406.200,-104.962,176.665,30.243,155.291
C04439=1080.077,405.954,-104.920,176.661,30.234,155.289
C04440=1080.071,405.708,-104.879,176.657,30.225,155.287
C04441=1080.064,405.460,-104.839,176.653,30.216,155.285
C04442=1080.057,405.215,-104.798,176.649,30.207,155.284
C04443=1080.050,404.968,-104.756,176.645,30.198,155.282
C04444=1080.044,404.721,-104.715,176.640,30.189,155.280
C04445=1080.037,404.475,-104.674,176.636,30.181,155.278
C04446=1080.030,404.228,-104.633,176.632,30.172,155.276
C04447=1080.023,403.982,-104.592,176.628,30.163,155.274
C04448=1080.017,403.734,-104.551,176.623,30.154,155.272
C04449=1080.010,403.489,-104.510,176.619,30.145,155.271
C04450=1080.003,403.242,-104.469,176.615,30.137,155.269
C04451=1079.997,402.995,-104.429,176.611,30.128,155.267
C04452=1079.989,402.749,-104.388,176.606,30.119,155.265
C04453=1079.983,402.502,-104.348,176.602,30.110,155.263
C04454=1079.976,402.256,-104.306,176.598,30.102,155.262
C04455=1079.969,402.009,-104.266,176.594,30.093,155.260
C04456=1079.962,401.762,-104.226,176.590,30.085,155.258
C04457=1079.956,401.516,-104.185,176.586,30.076,155.256
C04458=1079.949,401.270,-104.145,176.582,30.068,155.255
C04459=1079.942,401.023,-104.103,176.578,30.059,155.253
C04460=1079.936,400.776,-104.063,176.573,30.051,155.251
C04461=1079.929,400.529,-104.022,176.569,30.042,155.249
C04462=1079.923,400.282,-103.982,176.565,30.033,155.247
C04463=1079.916,400.037,-103.941,176.562,30.025,155.246
C04464=1079.909,399.789,-103.901,176.558,30.017,155.244
C04465=1079.903,399.551,-103.862,176.554,30.009,155.242
C04466=1079.897,399.310,-103.823,176.550,30.001,155.241
C04467=1079.890,399.071,-103.784,176.545,29.993,155.239
C04468=1079.884,398.831,-103.744,176.541,29.984,155.237
C04469=1079.877,398.591,-103.705,176.538,29.976,155.236
C04470=1079.871,398.352,-103.666,176.534,29.968,155.234
C04471=1079.864,398.112,-103.627,176.530,29.960,155.232
C04472=1079.857,397.873,-103.588,176.526,29.952,155.231
C04473=1079.851,397.626,-103.548,176.522,29.944,155.229
C04474=1079.844,397.379,-103.507,176.519,29.936,155.227
C04475=1079.838,397.132,-103.467,176.514,29.928,155.226
C04476=1079.831,396.886,-103.428,176.510,29.920,155.224
C04477=1079.824,396.640,-103.387,176.506,29.912,155.222
C04478=1079.818,396.393,-103.347,176.502,29.904,155.221
C04479=1079.811,396.146,-103.307,176.498,29.895,155.219
C04480=1079.805,395.899,-103.267,176.494,29.887,155.217
C04481=1079.798,395.653,-103.228,176.490,29.879,155.216
C04482=1079.791,395.406,-103.188,176.487,29.871,155.214
C04483=1079.785,395.160,-103.147,176.482,29.863,155.212
C04484=1079.779,394.913,-103.107,176.478,29.855,155.211
C04485=1079.772,394.666,-103.068,176.474,29.847,155.209
C04486=1079.765,394.419,-103.028,176.470,29.839,155.207
C04487=1079.758,394.172,-102.988,176.466,29.831,155.206
C04488=1079.752,393.926,-102.949,176.463,29.823,155.204
C04489=1079.745,393.679,-102.909,176.459,29.815,155.203
C04490=1079.739,393.433,-102.869,176.455,29.808,155.201
C04491=1079.732,393.186,-102.830,176.451,29.800,155.200
C04492=1079.726,392.939,-102.790,176.446,29.792,155.198
C04493=1079.719,392.692,-102.751,176.443,29.784,155.196
C04494=1079.712,392.446,-102.711,176.439,29.776,155.195
C04495=1079.706,392.199,-102.671,176.435,29.769,155.193
C04496=1079.699,391.953,-102.632,176.431,29.761,155.192
C04497=1079.693,391.705,-102.592,176.427,29.753,155.190
C04498=1079.686,391.459,-102.553,176.424,29.746,155.189
C04499=1079.680,391.212,-102.513,176.420,29.738,155.187
C04500=1079.673,390.966,-102.474,176.415,29.730,155.185
C04501=1079.666,390.719,-102.435,176.411,29.723,155.184
C04502=1079.660,390.472,-102.395,176.407,29.715,155.182
C04503=1079.653,390.226,-102.356,176.404,29.708,155.181
C04504=1079.646,389.979,-102.317,176.400,29.700,155.179
C04505=1079.640,389.732,-102.278,176.396,29.692,155.178
C04506=1079.633,389.485,-102.239,176.392,29.684,155.176
C04507=1079.626,389.239,-102.199,176.389,29.678,155.175
C04508=1079.620,388.992,-102.160,176.384,29.670,155.173
C04509=1079.613,388.745,-102.121,176.380,29.662,155.172
C04510=1079.606,388.498,-102.082,176.376,29.655,155.170
C04511=1079.601,388.252,-102.043,176.373,29.647,155.169
C04512=1079.594,388.005,-102.004,176.369,29.640,155.167
C04513=1079.587,387.758,-101.965,176.365,29.633,155.166
C04514=1079.581,387.511,-101.925,176.362,29.626,155.164
C04515=1079.574,387.265,-101.886,176.358,29.618,155.163
C04516=1079.567,387.018,-101.848,176.353,29.611,155.162
C04517=1079.560,386.771,-101.809,176.349,29.603,155.160
C04518=1079.555,386.525,-101.770,176.346,29.596,155.159
C04519=1079.548,386.278,-101.731,176.342,29.588,155.157
C04520=1079.541,386.031,-101.692,176.338,29.581,155.156
C04521=1079.536,385.799,-101.656,176.335,29.575,155.154
C04522=1079.530,385.566,-101.619,176.332,29.568,155.153
C04523=1079.524,385.334,-101.583,176.328,29.560,155.152
C04524=1079.517,385.101,-101.546,176.324,29.554,155.150
C04525=1079.512,384.868,-101.510,176.320,29.547,155.149
C04526=1079.505,384.636,-101.473,176.317,29.540,155.148
C04527=1079.500,384.403,-101.437,176.314,29.534,155.146
C04528=1079.493,384.172,-101.400,176.310,29.527,155.145
C04529=1079.487,383.924,-101.362,176.307,29.520,155.143
C04530=1079.481,383.677,-101.323,176.302,29.512,155.142
C04531=1079.474,383.430,-101.284,176.298,29.505,155.141
C04532=1079.468,383.184,-101.246,176.295,29.498,155.139
C04533=1079.461,382.937,-101.207,176.291,29.491,155.138
C04534=1079.455,382.691,-101.169,176.288,29.484,155.136
C04535=1079.449,382.443,-101.130,176.284,29.477,155.135
C04536=1079.442,382.196,-101.091,176.280,29.470,155.134
C04537=1079.436,381.949,-101.053,176.277,29.463,155.132
C04538=1079.430,381.703,-101.015,176.272,29.456,155.131
C04539=1079.423,381.455,-100.976,176.268,29.449,155.130
C04540=1079.417,381.209,-100.938,176.265,29.442,155.128
C04541=1079.410,380.962,-100.900,176.261,29.435,155.127
C04542=1079.404,380.715,-100.861,176.258,29.428,155.125
C04543=1079.397,380.468,-100.824,176.254,29.421,155.124
C04544=1079.390,380.221,-100.785,176.251,29.414,155.123
C04545=1079.384,379.974,-100.747,176.246,29.408,155.121
C04546=1079.378,379.727,-100.709,176.242,29.400,155.120
C04547=1079.371,379.480,-100.670,176.239,29.394,155.119
C04548=1079.365,379.234,-100.633,176.235,29.387,155.117
C04549=1079.358,378.986,-100.594,176.232,29.380,155.116
C04550=1079.352,378.739,-100.556,176.228,29.373,155.115
C04551=1079.346,378.493,-100.518,176.225,29.367,155.114
C04552=1079.339,378.246,-100.480,176.221,29.360,155.112
C04553=1079.333,377.999,-100.443,176.217,29.353,155.111
C04554=1079.326,377.751,-100.404,176.213,29.346,155.110
C04555=1079.320,377.505,-100.367,176.209,29.340,155.108
C04556=1079.313,377.258,-100.328,176.206,29.333,155.107
C04557=1079.307,377.011,-100.290,176.202,29.326,155.106
C04558=1079.301,376.764,-100.252,176.199,29.319,155.104
C04559=1079.294,376.517,-100.215,176.195,29.312,155.103
C04560=1079.288,376.270,-100.177,176.191,29.306,155.102
C04561=1079.282,376.023,-100.139,176.187,29.299,155.100
C04562=1079.275,375.776,-100.101,176.184,29.293,155.099
C04563=1079.270,375.529,-100.063,176.180,29.286,155.098
C04564=1079.263,375.282,-100.026,176.177,29.279,155.097
C04565=1079.256,375.035,-99.988,176.173,29.273,155.095
C04566=1079.250,374.788,-99.950,176.170,29.267,155.094
C04567=1079.244,374.541,-99.912,176.166,29.260,155.093
C04568=1079.238,374.293,-99.875,176.162,29.253,155.092
C04569=1079.232,374.047,-99.838,176.159,29.247,155.090
C04570=1079.225,373.800,-99.800,176.155,29.240,155.089
C04571=1079.219,373.553,-99.762,176.152,29.234,155.088
C04572=1079.213,373.306,-99.725,176.148,29.227,155.087
C04573=1079.206,373.058,-99.687,176.145,29.221,155.085
C04574=1079.200,372.812,-99.650,176.141,29.214,155.084
C04575=1079.193,372.564,-99.612,176.137,29.208,155.083
C04576=1079.187,372.318,-99.574,176.133,29.201,155.082
C04577=1079.182,372.099,-99.542,176.130,29.196,155.081
C04578=1079.175,371.881,-99.508,176.127,29.190,155.080
C04579=1079.171,371.663,-99.476,176.125,29.185,155.079
C04580=1079.165,371.445,-99.443,176.121,29.179,155.077
C04581=1079.159,371.227,-99.410,176.118,29.173,155.076
C04582=1079.153,371.009,-99.378,176.115,29.168,155.075
C04583=1079.148,370.791,-99.344,176.112,29.162,155.074
C04584=1079.143,370.573,-99.312,176.108,29.157,155.073
C04585=1079.135,370.326,-99.274,176.105,29.150,155.072
C04586=1079.130,370.078,-99.237,176.101,29.144,155.071
C04587=1079.123,369.832,-99.200,176.098,29.138,155.070
C04588=1079.117,369.584,-99.162,176.094,29.132,155.069
C04589=1079.110,369.338,-99.125,176.091,29.125,155.067
C04590=1079.105,369.090,-99.088,176.087,29.119,155.066
C04591=1079.098,368.843,-99.052,176.083,29.113,155.065
C04592=1079.092,368.596,-99.014,176.080,29.107,155.064
C04593=1079.085,368.349,-98.977,176.076,29.100,155.063
C04594=1079.080,368.101,-98.940,176.073,29.094,155.062
C04595=1079.073,367.855,-98.903,176.070,29.088,155.060
C04596=1079.067,367.608,-98.867,176.065,29.082,155.059
C04597=1079.061,367.360,-98.829,176.062,29.076,155.058
C04598=1079.054,367.113,-98.792,176.058,29.070,155.057
C04599=1079.048,366.866,-98.755,176.055,29.063,155.056
C04600=1079.042,366.619,-98.718,176.052,29.057,155.055
C04601=1079.036,366.372,-98.682,176.048,29.051,155.053
C04602=1079.030,366.124,-98.645,176.045,29.045,155.052
C04603=1079.023,365.877,-98.607,176.041,29.039,155.051
C04604=1079.017,365.630,-98.570,176.037,29.033,155.050
C04605=1079.011,365.383,-98.534,176.034,29.027,155.049
C04606=1079.005,365.136,-98.498,176.031,29.020,155.048
C04607=1078.999,364.888,-98.460,176.027,29.015,155.047
C04608=1078.993,364.641,-98.424,176.024,29.009,155.045
C04609=1078.986,364.394,-98.388,176.021,29.002,155.044
C04610=1078.979,364.147,-98.351,176.016,28.997,155.043
C04611=1078.973,363.900,-98.314,176.013,28.991,155.042
C04612=1078.968,363.652,-98.277,176.010,28.985,155.041
C04613=1078.961,363.405,-98.241,176.006,28.979,155.040
C04614=1078.955,363.158,-98.204,176.003,28.973,155.039
C04615=1078.948,362.911,-98.168,176.000,28.967,155.038
C04616=1078.942,362.664,-98.132,175.995,28.961,155.037
C04617=1078.936,362.417,-98.095,175.992,28.955,155.036
C04618=1078.930,362.169,-98.059,175.989,28.949,155.034
C04619=1078.923,361.922,-98.023,175.985,28.943,155.033
C04620=1078.918,361.675,-97.986,175.982,28.937,155.032
C04621=1078.911,361.427,-97.949,175.979,28.932,155.031
C04622=1078.905,361.180,-97.913,175.975,28.926,155.030
C04623=1078.899,360.932,-97.877,175.971,28.920,155.029
C04624=1078.892,360.685,-97.840,175.968,28.914,155.028
C04625=1078.886,360.438,-97.804,175.965,28.908,155.027
C04626=1078.880,360.191,-97.768,175.961,28.902,155.026
C04627=1078.874,359.943,-97.732,175.958,28.896,155.025
C04628=1078.867,359.696,-97.695,175.954,28.891,155.024
C04629=1078.861,359.449,-97.660,175.951,28.885,155.023
C04630=1078.855,359.202,-97.623,175.947,28.879,155.022
C04631=1078.848,358.955,-97.587,175.944,28.873,155.021
C04632=1078.842,358.707,-97.551,175.941,28.868,155.020
C04633=1078.838,358.498,-97.520,175.937,28.863,155.019
C04634=1078.832,358.288,-97.490,175.935,28.858,155.018
C04635=1078.827,358.077,-97.459,175.932,28.853,155.017
C04636=1078.821,357.867,-97.429,175.929,28.848,155.016
C04637=1078.816,357.657,-97.398,175.926,28.843,155.015
C04638=1078.810,357.448,-97.367,175.923,28.839,155.014
C04639=1078.806,357.238,-97.337,175.921,28.834,155.013
C04640=1078.801,357.028,-97.306,175.917,28.829,155.013
C04641=1078.794,356.780,-97.271,175.914,28.824,155.012
C04642=1078.788,356.533,-97.235,175.911,28.818,155.010
C04643=1078.782,356.285,-97.199,175.907,28.812,155.009
C04644=1078.775,356.038,-97.163,175.904,28.807,155.008
C04645=1078.769,355.791,-97.127,175.900,28.801,155.007
C04646=1078.763,355.543,-97.091,175.897,28.795,155.006
C04647=1078.758,355.297,-97.055,175.894,28.790,155.005
C04648=1078.751,355.049,-97.020,175.890,28.784,155.004
C04649=1078.745,354.802,-96.984,175.887,28.778,155.003
C04650=1078.739,354.554,-96.948,175.884,28.773,155.002
C04651=1078.732,354.307,-96.912,175.880,28.768,155.001
C04652=1078.726,354.059,-96.876,175.877,28.762,155.000
C04653=1078.721,353.812,-96.841,175.873,28.756,154.999
C04654=1078.714,353.565,-96.806,175.870,28.750,154.998
C04655=1078.708,353.317,-96.770,175.867,28.745,154.997
C04656=1078.702,353.070,-96.734,175.864,28.740,154.996
C04657=1078.696,352.822,-96.699,175.860,28.734,154.995
C04658=1078.690,352.576,-96.663,175.856,28.729,154.994
C04659=1078.684,352.328,-96.627,175.853,28.723,154.993
C04660=1078.678,352.080,-96.592,175.850,28.718,154.992
C04661=1078.671,351.833,-96.557,175.847,28.712,154.991
C04662=1078.665,351.585,-96.521,175.843,28.707,154.990
C04663=1078.659,351.338,-96.485,175.840,28.702,154.990
C04664=1078.653,351.091,-96.450,175.836,28.696,154.989
C04665=1078.646,350.843,-96.415,175.833,28.691,154.988
C04666=1078.640,350.596,-96.379,175.830,28.685,154.987
C04667=1078.635,350.348,-96.345,175.827,28.680,154.986
C04668=1078.629,350.101,-96.309,175.823,28.674,154.985
C04669=1078.622,349.853,-96.274,175.820,28.669,154.984
C04670=1078.616,349.606,-96.238,175.817,28.664,154.983
C04671=1078.610,349.359,-96.203,175.813,28.658,154.982
C04672=1078.604,349.111,-96.168,175.810,28.653,154.981
C04673=1078.597,348.864,-96.133,175.806,28.647,154.980
C04674=1078.592,348.616,-96.098,175.803,28.642,154.979
C04675=1078.585,348.369,-96.063,175.800,28.637,154.978
C04676=1078.579,348.121,-96.027,175.797,28.632,154.977
C04677=1078.573,347.875,-95.992,175.794,28.626,154.976
C04678=1078.567,347.626,-95.957,175.790,28.621,154.975
C04679=1078.560,347.379,-95.922,175.786,28.616,154.974
C04680=1078.555,347.132,-95.887,175.783,28.610,154.973
C04681=1078.548,346.884,-95.852,175.780,28.605,154.972
C04682=1078.542,346.636,-95.817,175.777,28.600,154.972
C04683=1078.536,346.390,-95.782,175.774,28.595,154.971
C04684=1078.530,346.141,-95.747,175.770,28.590,154.970
C04685=1078.524,345.895,-95.712,175.767,28.584,154.969
C04686=1078.519,345.647,-95.677,175.764,28.579,154.968
C04687=1078.512,345.399,-95.642,175.761,28.574,154.967
C04688=1078.506,345.152,-95.608,175.758,28.569,154.966
C04689=1078.496,344.736,-95.549,175.752,28.560,154.964
C04690=1078.485,344.318,-95.490,175.746,28.551,154.963
C04691=1078.475,343.902,-95.432,175.741,28.542,154.961
C04692=1078.465,343.485,-95.373,175.735,28.534,154.960
C04693=1078.459,343.237,-95.338,175.732,28.528,154.959
C04694=1078.453,342.990,-95.304,175.729,28.523,154.958
C04695=1078.447,342.742,-95.268,175.725,28.518,154.957
C04696=1078.440,342.494,-95.234,175.722,28.513,154.956
C04697=1078.434,342.247,-95.200,175.719,28.508,154.956
C04698=1078.428,341.999,-95.166,175.716,28.503,154.955
C04699=1078.422,341.752,-95.131,175.713,28.498,154.954
C04700=1078.416,341.504,-95.096,175.709,28.493,154.953
C04701=1078.410,341.257,-95.062,175.706,28.488,154.952
C04702=1078.404,341.009,-95.027,175.703,28.483,154.951
C04703=1078.398,340.762,-94.993,175.700,28.478,154.950
C04704=1078.391,340.514,-94.958,175.696,28.473,154.949
C04705=1078.386,340.267,-94.923,175.693,28.468,154.948
C04706=1078.380,340.019,-94.889,175.690,28.463,154.948
C04707=1078.374,339.771,-94.855,175.687,28.457,154.947
C04708=1078.368,339.524,-94.821,175.684,28.453,154.946
C04709=1078.361,339.276,-94.787,175.680,28.448,154.945
C04710=1078.355,339.029,-94.752,175.677,28.442,154.944
C04711=1078.349,338.781,-94.717,175.674,28.438,154.943
C04712=1078.344,338.534,-94.683,175.671,28.433,154.942
C04713=1078.338,338.286,-94.649,175.668,28.427,154.942
C04714=1078.331,338.038,-94.614,175.664,28.422,154.941
C04715=1078.325,337.791,-94.580,175.661,28.418,154.940
C04716=1078.319,337.543,-94.546,175.658,28.412,154.939
C04717=1078.313,337.295,-94.512,175.655,28.408,154.938
C04718=1078.308,337.048,-94.478,175.652,28.403,154.937
C04719=1078.301,336.800,-94.444,175.648,28.398,154.936
C04720=1078.295,336.553,-94.410,175.645,28.393,154.936
C04721=1078.289,336.305,-94.375,175.642,28.388,154.935
C04722=1078.283,336.057,-94.341,175.639,28.383,154.934
C04723=1078.277,335.810,-94.307,175.636,28.378,154.933
C04724=1078.271,335.562,-94.273,175.632,28.373,154.932
C04725=1078.265,335.314,-94.240,175.629,28.368,154.931
C04726=1078.258,335.067,-94.206,175.626,28.363,154.931
C04727=1078.252,334.819,-94.172,175.623,28.359,154.930
C04728=1078.246,334.572,-94.138,175.619,28.354,154.929
C04729=1078.241,334.324,-94.104,175.616,28.349,154.928
C04730=1078.234,334.076,-94.070,175.613,28.344,154.927
C04731=1078.228,333.829,-94.036,175.610,28.339,154.926
C04732=1078.223,333.581,-94.003,175.607,28.334,154.926
C04733=1078.217,333.334,-93.968,175.603,28.330,154.925
C04734=1078.210,333.086,-93.934,175.600,28.324,154.924
C04735=1078.205,332.838,-93.901,175.597,28.320,154.923
C04736=1078.198,332.591,-93.867,175.595,28.315,154.922
C04737=1078.192,332.344,-93.833,175.592,28.310,154.922
C04738=1078.186,332.095,-93.800,175.588,28.306,154.921
C04739=1078.180,331.848,-93.765,175.585,28.301,154.920
C04740=1078.175,331.600,-93.732,175.582,28.296,154.919
C04741=1078.169,331.389,-93.703,175.580,28.292,154.918
C04742=1078.163,331.178,-93.675,175.576,28.288,154.918
C04743=1078.158,330.966,-93.646,175.574,28.284,154.917
C04744=1078.154,330.756,-93.618,175.571,28.280,154.916
C04745=1078.149,330.544,-93.589,175.568,28.276,154.916
C04746=1078.143,330.334,-93.561,175.566,28.272,154.915
C04747=1078.137,330.123,-93.532,175.563,28.268,154.914
C04748=1078.133,329.911,-93.503,175.560,28.264,154.914
C04749=1078.126,329.664,-93.470,175.557,28.259,154.913
C04750=1078.120,329.416,-93.437,175.554,28.254,154.912
C04751=1078.114,329.168,-93.403,175.551,28.250,154.911
C04752=1078.108,328.921,-93.369,175.548,28.245,154.911
C04753=1078.102,328.673,-93.336,175.545,28.241,154.910
C04754=1078.096,328.425,-93.303,175.542,28.236,154.909
C04755=1078.089,328.177,-93.269,175.538,28.231,154.908
C04756=1078.083,327.930,-93.236,175.535,28.227,154.908
C04757=1078.077,327.682,-93.203,175.532,28.222,154.907
C04758=1078.071,327.434,-93.170,175.529,28.217,154.906
C04759=1078.065,327.187,-93.136,175.526,28.212,154.905
C04760=1078.059,326.939,-93.103,175.523,28.208,154.904
C04761=1078.053,326.691,-93.070,175.520,28.203,154.904
C04762=1078.047,326.443,-93.037,175.517,28.199,154.903
C04763=1078.041,326.195,-93.004,175.514,28.194,154.902
C04764=1078.034,325.948,-92.970,175.510,28.190,154.902
C04765=1078.029,325.700,-92.937,175.507,28.185,154.901
C04766=1078.023,325.453,-92.904,175.504,28.180,154.900
C04767=1078.017,325.205,-92.871,175.502,28.176,154.899
C04768=1078.011,324.957,-92.838,175.498,28.171,154.898
C04769=1078.005,324.709,-92.805,175.495,28.167,154.898
C04770=1077.999,324.462,-92.772,175.492,28.162,154.897
C04771=1077.993,324.214,-92.739,175.489,28.157,154.896
C04772=1077.986,323.965,-92.705,175.485,28.153,154.895
C04773=1077.980,323.718,-92.673,175.483,28.149,154.895
C04774=1077.975,323.470,-92.639,175.480,28.144,154.894
C04775=1077.968,323.222,-92.607,175.477,28.139,154.893
C04776=1077.963,322.974,-92.573,175.474,28.134,154.892
C04777=1077.956,322.727,-92.541,175.470,28.130,154.892
C04778=1077.950,322.479,-92.508,175.468,28.126,154.891
C04779=1077.945,322.231,-92.474,175.465,28.121,154.890
C04780=1077.938,321.984,-92.442,175.462,28.116,154.889
C04781=1077.933,321.736,-92.408,175.458,28.112,154.889
C04782=1077.927,321.488,-92.377,175.455,28.107,154.888
C04783=1077.921,321.241,-92.344,175.452,28.103,154.887
C04784=1077.916,320.993,-92.311,175.450,28.098,154.886
C04785=1077.909,320.745,-92.278,175.446,28.094,154.886
C04786=1077.903,320.498,-92.245,175.443,28.089,154.885
C04787=1077.897,320.250,-92.212,175.440,28.085,154.884
C04788=1077.891,320.002,-92.180,175.438,28.080,154.883
C04789=1077.885,319.754,-92.147,175.435,28.076,154.883
C04790=1077.880,319.506,-92.114,175.431,28.071,154.882
C04791=1077.873,319.258,-92.081,175.428,28.067,154.881
C04792=1077.867,319.010,-92.049,175.425,28.062,154.880
C04793=1077.862,318.763,-92.016,175.423,28.058,154.880
C04794=1077.856,318.515,-91.983,175.419,28.053,154.879
C04795=1077.850,318.267,-91.951,175.416,28.049,154.878
C04796=1077.844,318.019,-91.918,175.413,28.044,154.877
C04797=1077.839,317.805,-91.890,175.411,28.040,154.877
C04798=1077.834,317.590,-91.862,175.408,28.036,154.876
C04799=1077.829,317.376,-91.833,175.406,28.033,154.876
C04800=1077.824,317.162,-91.805,175.403,28.029,154.875
C04801=1077.819,316.948,-91.778,175.400,28.025,154.874
C04802=1077.814,316.734,-91.749,175.398,28.021,154.874
C04803=1077.810,316.519,-91.721,175.395,28.017,154.873
C04804=1077.804,316.305,-91.693,175.392,28.013,154.872
C04805=1077.798,316.057,-91.660,175.390,28.009,154.872
C04806=1077.792,315.808,-91.628,175.387,28.004,154.871
C04807=1077.787,315.562,-91.596,175.384,28.000,154.870
C04808=1077.781,315.313,-91.564,175.380,27.995,154.869
C04809=1077.775,315.065,-91.530,175.378,27.991,154.869
C04810=1077.770,314.818,-91.499,175.375,27.986,154.868
C04811=1077.764,314.570,-91.466,175.372,27.982,154.867
C04812=1077.758,314.322,-91.434,175.368,27.977,154.867
C04813=1077.752,314.074,-91.402,175.366,27.973,154.866
C04814=1077.745,313.826,-91.369,175.363,27.969,154.865
C04815=1077.739,313.578,-91.338,175.360,27.965,154.865
C04816=1077.733,313.331,-91.306,175.357,27.961,154.864
C04817=1077.727,313.083,-91.273,175.354,27.956,154.863
C04818=1077.721,312.835,-91.241,175.351,27.952,154.862
C04819=1077.715,312.587,-91.209,175.348,27.947,154.862
C04820=1077.709,312.339,-91.177,175.345,27.943,154.861
C04821=1077.702,312.092,-91.145,175.342,27.939,154.861
C04822=1077.697,311.844,-91.113,175.339,27.935,154.860
C04823=1077.691,311.596,-91.081,175.336,27.930,154.859
C04824=1077.684,311.348,-91.049,175.333,27.926,154.858
C04825=1077.679,311.101,-91.017,175.330,27.922,154.858
C04826=1077.672,310.853,-90.986,175.327,27.917,154.857
C04827=1077.666,310.604,-90.954,175.324,27.913,154.856
C04828=1077.660,310.356,-90.921,175.321,27.909,154.856
C04829=1077.655,310.109,-90.890,175.318,27.905,154.855
C04830=1077.649,309.861,-90.858,175.315,27.900,154.854
C04831=1077.642,309.613,-90.826,175.312,27.896,154.854
C04832=1077.636,309.366,-90.794,175.309,27.892,154.853
C04833=1077.630,309.118,-90.762,175.306,27.888,154.852
C04834=1077.624,308.869,-90.730,175.304,27.884,154.852
C04835=1077.618,308.622,-90.699,175.300,27.879,154.851
C04836=1077.612,308.374,-90.667,175.297,27.875,154.850
C04837=1077.606,308.126,-90.635,175.295,27.871,154.850
C04838=1077.601,307.878,-90.603,175.292,27.867,154.849
C04839=1077.594,307.630,-90.572,175.288,27.862,154.848
C04840=1077.589,307.383,-90.540,175.286,27.858,154.848
C04841=1077.583,307.135,-90.508,175.283,27.854,154.847
C04842=1077.576,306.887,-90.477,175.280,27.850,154.846
C04843=1077.571,306.638,-90.446,175.277,27.846,154.846
C04844=1077.565,306.390,-90.414,175.274,27.841,154.845
C04845=1077.559,306.143,-90.383,175.271,27.837,154.844
C04846=1077.553,305.895,-90.351,175.268,27.832,154.844
C04847=1077.548,305.647,-90.319,175.265,27.829,154.843
C04848=1077.542,305.399,-90.287,175.262,27.824,154.842
C04849=1077.535,305.152,-90.256,175.259,27.820,154.842
C04850=1077.530,304.903,-90.224,175.257,27.816,154.841
C04851=1077.524,304.656,-90.193,175.253,27.811,154.840
C04852=1077.518,304.408,-90.161,175.251,27.807,154.840
C04853=1077.513,304.195,-90.134,175.248,27.804,154.839
C04854=1077.507,303.982,-90.107,175.245,27.800,154.839
C04855=1077.503,303.769,-90.080,175.243,27.796,154.838
C04856=1077.498,303.557,-90.054,175.241,27.793,154.837
C04857=1077.493,303.344,-90.026,175.238,27.789,154.837
C04858=1077.487,303.131,-90.000,175.236,27.786,154.836
C04859=1077.483,302.918,-89.973,175.234,27.782,154.836
C04860=1077.478,302.706,-89.946,175.231,27.779,154.835
C04861=1077.472,302.457,-89.914,175.228,27.774,154.834
C04862=1077.466,302.210,-89.883,175.225,27.770,154.834
C04863=1077.460,301.962,-89.851,175.223,27.766,154.833
C04864=1077.455,301.714,-89.820,175.219,27.762,154.832
C04865=1077.448,301.466,-89.789,175.216,27.757,154.832
C04866=1077.443,301.218,-89.758,175.214,27.753,154.831
C04867=1077.438,300.970,-89.726,175.211,27.749,154.830
C04868=1077.431,300.722,-89.695,175.208,27.745,154.830
C04869=1077.426,300.474,-89.664,175.205,27.741,154.829
C04870=1077.420,300.227,-89.633,175.202,27.736,154.828
C04871=1077.414,299.978,-89.602,175.200,27.732,154.828
C04872=1077.408,299.731,-89.570,175.196,27.728,154.827
C04873=1077.402,299.482,-89.539,175.193,27.724,154.827
C04874=1077.397,299.235,-89.507,175.191,27.720,154.826
C04875=1077.391,298.987,-89.477,175.188,27.715,154.825
C04876=1077.386,298.739,-89.446,175.185,27.711,154.824
C04877=1077.379,298.491,-89.415,175.182,27.707,154.824
C04878=1077.374,298.243,-89.384,175.180,27.703,154.823
C04879=1077.368,297.996,-89.353,175.177,27.699,154.823
C04880=1077.362,297.747,-89.321,175.173,27.695,154.822
C04881=1077.356,297.499,-89.291,175.171,27.691,154.821
C04882=1077.350,297.252,-89.260,175.168,27.686,154.821
C04883=1077.345,297.003,-89.229,175.166,27.682,154.820
C04884=1077.339,296.755,-89.198,175.162,27.678,154.819
C04885=1077.333,296.508,-89.167,175.159,27.674,154.819
C04886=1077.327,296.259,-89.136,175.157,27.670,154.818
C04887=1077.321,296.011,-89.106,175.154,27.666,154.817
C04888=1077.315,295.763,-89.075,175.151,27.662,154.817
C04889=1077.310,295.515,-89.044,175.148,27.658,154.816
C04890=1077.304,295.267,-89.013,175.146,27.654,154.816
C04891=1077.298,295.020,-88.983,175.143,27.650,154.815
C04892=1077.291,294.771,-88.952,175.139,27.645,154.814
C04893=1077.286,294.523,-88.921,175.137,27.642,154.814
C04894=1077.281,294.275,-88.891,175.134,27.638,154.813
C04895=1077.274,294.027,-88.860,175.131,27.634,154.812
C04896=1077.268,293.779,-88.829,175.128,27.629,154.812
C04897=1077.262,293.531,-88.798,175.126,27.625,154.811
C04898=1077.256,293.284,-88.768,175.123,27.621,154.810
C04899=1077.250,293.035,-88.737,175.120,27.618,154.810
C04900=1077.245,292.787,-88.706,175.117,27.613,154.809
C04901=1077.239,292.539,-88.676,175.114,27.609,154.809
C04902=1077.233,292.291,-88.646,175.112,27.605,154.808
C04903=1077.227,292.043,-88.615,175.108,27.601,154.807
C04904=1077.221,291.795,-88.585,175.106,27.597,154.807
C04905=1077.215,291.547,-88.554,175.103,27.593,154.806
C04906=1077.209,291.299,-88.524,175.101,27.589,154.806
C04907=1077.204,291.051,-88.493,175.097,27.585,154.805
C04908=1077.198,290.803,-88.462,175.095,27.581,154.804
C04909=1077.188,290.392,-88.412,175.090,27.575,154.803
C04910=1077.178,289.980,-88.362,175.086,27.568,154.802
C04911=1077.169,289.570,-88.312,175.081,27.561,154.801
C04912=1077.159,289.159,-88.261,175.076,27.554,154.800
C04913=1077.153,288.911,-88.231,175.074,27.551,154.800
C04914=1077.147,288.662,-88.201,175.070,27.546,154.799
C04915=1077.141,288.414,-88.171,175.068,27.543,154.798
C04916=1077.135,288.166,-88.141,175.065,27.539,154.798
C04917=1077.129,287.919,-88.111,175.063,27.535,154.797
C04918=1077.124,287.670,-88.081,175.059,27.530,154.797
C04919=1077.118,287.422,-88.051,175.057,27.527,154.796
C04920=1077.111,287.174,-88.020,175.054,27.523,154.795
C04921=1077.105,286.926,-87.990,175.052,27.519,154.795
C04922=1077.100,286.677,-87.960,175.048,27.515,154.794
C04923=1077.094,286.430,-87.930,175.046,27.511,154.794
C04924=1077.088,286.182,-87.899,175.043,27.507,154.793
C04925=1077.082,285.934,-87.870,175.041,27.503,154.792
C04926=1077.076,285.686,-87.840,175.037,27.499,154.792
C04927=1077.071,285.437,-87.810,175.035,27.495,154.791
C04928=1077.064,285.189,-87.779,175.032,27.491,154.791
C04929=1077.059,284.940,-87.750,175.030,27.487,154.790
C04930=1077.053,284.693,-87.719,175.026,27.483,154.789
C04931=1077.047,284.445,-87.689,175.024,27.479,154.789
C04932=1077.041,284.197,-87.660,175.021,27.475,154.788
C04933=1077.035,283.949,-87.630,175.018,27.472,154.788
C04934=1077.030,283.700,-87.600,175.016,27.468,154.787
C04935=1077.024,283.453,-87.570,175.013,27.463,154.786
C04936=1077.018,283.204,-87.540,175.011,27.460,154.786
C04937=1077.012,282.956,-87.510,175.007,27.456,154.785
C04938=1077.006,282.708,-87.481,175.005,27.452,154.785
C04939=1077.001,282.460,-87.451,175.002,27.448,154.784
C04940=1076.995,282.212,-87.421,175.000,27.444,154.783
C04941=1076.989,281.964,-87.391,174.996,27.440,154.783
C04942=1076.984,281.716,-87.361,174.994,27.436,154.782
C04943=1076.977,281.468,-87.332,174.991,27.432,154.782
C04944=1076.972,281.219,-87.302,174.989,27.428,154.781
C04945=1076.966,280.971,-87.272,174.986,27.424,154.780
C04946=1076.960,280.723,-87.242,174.983,27.420,154.780
C04947=1076.954,280.475,-87.213,174.981,27.416,154.779
C04948=1076.948,280.227,-87.183,174.978,27.412,154.779
C04949=1076.943,279.978,-87.153,174.975,27.409,154.778
C04950=1076.937,279.730,-87.124,174.972,27.404,154.777
C04951=1076.931,279.482,-87.094,174.970,27.401,154.777
C04952=1076.925,279.234,-87.065,174.967,27.397,154.776
C04953=1076.919,278.986,-87.035,174.964,27.393,154.776
C04954=1076.914,278.738,-87.005,174.962,27.389,154.775
C04955=1076.907,278.489,-86.976,174.959,27.385,154.775
C04956=1076.902,278.241,-86.947,174.956,27.381,154.774
C04957=1076.896,277.993,-86.918,174.953,27.377,154.773
C04958=1076.890,277.745,-86.887,174.951,27.373,154.773
C04959=1076.883,277.497,-86.858,174.948,27.370,154.772
C04960=1076.878,277.248,-86.829,174.945,27.366,154.772
C04961=1076.869,276.848,-86.781,174.942,27.360,154.771
C04962=1076.859,276.446,-86.734,174.937,27.353,154.770
C04963=1076.850,276.045,-86.687,174.932,27.347,154.769
C04964=1076.841,275.644,-86.639,174.928,27.340,154.768
C04965=1076.835,275.395,-86.610,174.926,27.337,154.767
C04966=1076.829,275.147,-86.580,174.923,27.333,154.767
C04967=1076.823,274.900,-86.552,174.920,27.329,154.766
C04968=1076.818,274.651,-86.522,174.917,27.325,154.765
C04969=1076.812,274.403,-86.493,174.915,27.321,154.765
C04970=1076.806,274.155,-86.463,174.913,27.317,154.764
C04971=1076.800,273.906,-86.434,174.909,27.313,154.764
C04972=1076.794,273.658,-86.405,174.907,27.309,154.763
C04973=1076.787,273.345,-86.368,174.904,27.305,154.762
C04974=1076.779,273.030,-86.331,174.900,27.300,154.762
C04975=1076.772,272.717,-86.295,174.897,27.295,154.761
C04976=1076.764,272.402,-86.258,174.894,27.290,154.760
C04977=1076.758,272.154,-86.229,174.891,27.286,154.760
C04978=1076.753,271.905,-86.199,174.888,27.283,154.759
C04979=1076.747,271.657,-86.171,174.886,27.279,154.759
C04980=1076.741,271.409,-86.142,174.883,27.275,154.758
C04981=1076.736,271.160,-86.112,174.881,27.271,154.757
C04982=1076.729,270.912,-86.083,174.877,27.267,154.757
C04983=1076.723,270.664,-86.055,174.875,27.263,154.756
C04984=1076.718,270.416,-86.026,174.873,27.259,154.756
C04985=1076.712,270.168,-85.997,174.870,27.256,154.755
C04986=1076.706,269.919,-85.968,174.867,27.252,154.755
C04987=1076.700,269.671,-85.939,174.865,27.248,154.754
C04988=1076.695,269.423,-85.910,174.862,27.244,154.753
C04989=1076.689,269.174,-85.882,174.860,27.240,154.753
C04990=1076.683,268.926,-85.853,174.856,27.236,154.752
C04991=1076.677,268.678,-85.824,174.854,27.233,154.752
C04992=1076.671,268.429,-85.795,174.852,27.229,154.751
C04993=1076.666,268.182,-85.766,174.848,27.225,154.751
C04994=1076.660,267.933,-85.738,174.846,27.221,154.750
C04995=1076.654,267.685,-85.709,174.844,27.217,154.749
C04996=1076.648,267.436,-85.680,174.841,27.214,154.749
C04997=1076.642,267.188,-85.652,174.838,27.210,154.748
C04998=1076.636,266.940,-85.623,174.836,27.206,154.748
C04999=1076.631,266.691,-85.594,174.833,27.202,154.747
C05000=1076.625,266.444,-85.565,174.831,27.198,154.747
C05001=1076.619,266.195,-85.537,174.828,27.195,154.746
C05002=1076.613,265.946,-85.508,174.825,27.190,154.745
C05003=1076.607,265.699,-85.480,174.823,27.187,154.745
C05004=1076.601,265.450,-85.451,174.821,27.183,154.744
C05005=1076.595,265.202,-85.422,174.817,27.179,154.744
C05006=1076.590,264.954,-85.394,174.815,27.176,154.743
C05007=1076.584,264.706,-85.365,174.813,27.172,154.743
C05008=1076.578,264.457,-85.337,174.810,27.168,154.742
C05009=1076.573,264.209,-85.309,174.807,27.164,154.741
C05010=1076.567,263.961,-85.280,174.805,27.160,154.741
C05011=1076.561,263.712,-85.251,174.802,27.156,154.740
C05012=1076.555,263.463,-85.223,174.800,27.153,154.740
C05013=1076.547,263.131,-85.185,174.796,27.148,154.739
C05014=1076.539,262.800,-85.147,174.793,27.143,154.738
C05015=1076.531,262.468,-85.110,174.789,27.138,154.738
C05016=1076.523,262.136,-85.072,174.785,27.133,154.737
C05017=1076.517,261.887,-85.044,174.783,27.129,154.736
C05018=1076.511,261.639,-85.015,174.781,27.125,154.736
C05019=1076.505,261.391,-84.987,174.778,27.121,154.735
C05020=1076.499,261.142,-84.958,174.775,27.118,154.735
C05021=1076.493,260.894,-84.931,174.773,27.114,154.734
C05022=1076.487,260.646,-84.903,174.771,27.110,154.734
C05023=1076.481,260.397,-84.874,174.768,27.106,154.733
C05024=1076.476,260.148,-84.846,174.765,27.103,154.732
C05025=1076.470,259.901,-84.817,174.763,27.099,154.732
C05026=1076.463,259.652,-84.790,174.760,27.096,154.731
C05027=1076.458,259.404,-84.762,174.758,27.092,154.731
C05028=1076.452,259.156,-84.733,174.755,27.088,154.730
C05029=1076.446,258.907,-84.705,174.752,27.084,154.730
C05030=1076.441,258.659,-84.677,174.750,27.081,154.729
C05031=1076.434,258.410,-84.649,174.748,27.077,154.729
C05032=1076.429,258.162,-84.621,174.745,27.073,154.728
C05033=1076.423,257.914,-84.593,174.742,27.069,154.728
C05034=1076.417,257.666,-84.565,174.740,27.065,154.727
C05035=1076.411,257.417,-84.537,174.738,27.062,154.726
C05036=1076.405,257.169,-84.510,174.735,27.058,154.726
C05037=1076.399,256.920,-84.481,174.732,27.054,154.725
C05038=1076.393,256.672,-84.453,174.730,27.050,154.725
C05039=1076.387,256.424,-84.426,174.727,27.047,154.724
C05040=1076.381,256.175,-84.397,174.724,27.043,154.724
C05041=1076.376,255.926,-84.370,174.722,27.039,154.723
C05042=1076.370,255.678,-84.342,174.720,27.035,154.723
C05043=1076.364,255.430,-84.314,174.717,27.032,154.722
C05044=1076.358,255.181,-84.286,174.714,27.028,154.721
C05045=1076.353,254.933,-84.258,174.712,27.024,154.721
C05046=1076.347,254.685,-84.231,174.710,27.020,154.720
C05047=1076.341,254.437,-84.202,174.707,27.017,154.720
C05048=1076.336,254.188,-84.175,174.704,27.012,154.719
C05049=1076.329,253.940,-84.147,174.702,27.009,154.719
C05050=1076.324,253.691,-84.119,174.700,27.005,154.718
C05051=1076.318,253.443,-84.091,174.697,27.002,154.718
C05052=1076.312,253.194,-84.064,174.694,26.997,154.717
C05053=1076.306,252.946,-84.036,174.692,26.994,154.716
C05054=1076.301,252.698,-84.008,174.690,26.990,154.716
C05055=1076.295,252.450,-83.981,174.688,26.986,154.715
C05056=1076.289,252.200,-83.953,174.684,26.982,154.715
C05057=1076.284,251.952,-83.925,174.682,26.979,154.714
C05058=1076.277,251.704,-83.897,174.680,26.975,154.714
C05059=1076.272,251.455,-83.870,174.678,26.971,154.713
C05060=1076.267,251.207,-83.842,174.675,26.968,154.713
C05061=1076.260,250.959,-83.814,174.672,26.963,154.712
C05062=1076.255,250.710,-83.787,174.670,26.960,154.711
C05063=1076.250,250.462,-83.759,174.668,26.956,154.711
C05064=1076.243,250.213,-83.732,174.665,26.952,154.710
C05065=1076.234,249.813,-83.687,174.661,26.946,154.709
C05066=1076.225,249.413,-83.644,174.657,26.940,154.708
C05067=1076.217,249.012,-83.599,174.653,26.934,154.707
C05068=1076.207,248.611,-83.554,174.649,26.928,154.707
C05069=1076.201,248.363,-83.527,174.647,26.924,154.706
C05070=1076.196,248.114,-83.500,174.645,26.920,154.705
C05071=1076.190,247.866,-83.472,174.642,26.917,154.705
C05072=1076.185,247.617,-83.445,174.639,26.912,154.704
C05073=1076.179,247.368,-83.417,174.637,26.909,154.704
C05074=1076.173,247.120,-83.390,174.635,26.905,154.703
C05075=1076.168,246.872,-83.363,174.633,26.901,154.703
C05076=1076.162,246.624,-83.335,174.629,26.897,154.702
C05077=1076.155,246.375,-83.308,174.627,26.894,154.702
C05078=1076.150,246.126,-83.281,174.625,26.890,154.701
C05079=1076.144,245.878,-83.254,174.623,26.886,154.700
C05080=1076.139,245.629,-83.226,174.620,26.883,154.700
C05081=1076.133,245.381,-83.199,174.617,26.879,154.699
C05082=1076.127,245.133,-83.172,174.615,26.875,154.699
C05083=1076.122,244.884,-83.145,174.613,26.871,154.698
C05084=1076.115,244.635,-83.118,174.611,26.868,154.698
C05085=1076.109,244.388,-83.090,174.608,26.864,154.697
C05086=1076.104,244.139,-83.063,174.606,26.860,154.697
C05087=1076.099,243.890,-83.037,174.603,26.856,154.696
C05088=1076.092,243.641,-83.010,174.601,26.853,154.696
C05089=1076.087,243.393,-82.982,174.598,26.849,154.695
C05090=1076.081,243.145,-82.955,174.596,26.845,154.694
C05091=1076.076,242.896,-82.928,174.594,26.841,154.694
C05092=1076.070,242.648,-82.901,174.591,26.837,154.693
C05093=1076.064,242.399,-82.874,174.589,26.834,154.693
C05094=1076.058,242.151,-82.847,174.586,26.830,154.692
C05095=1076.052,241.903,-82.820,174.584,26.826,154.692
C05096=1076.046,241.654,-82.793,174.582,26.823,154.691
C05097=1076.041,241.405,-82.766,174.580,26.819,154.690
C05098=1076.035,241.157,-82.739,174.577,26.815,154.690
C05099=1076.029,240.908,-82.712,174.574,26.811,154.689
C05100=1076.023,240.660,-82.686,174.572,26.808,154.689
C05101=1076.017,240.412,-82.659,174.570,26.804,154.688
C05102=1076.011,240.163,-82.632,174.567,26.800,154.688
C05103=1076.005,239.914,-82.606,174.565,26.797,154.687
C05104=1076.000,239.666,-82.578,174.563,26.793,154.687
C05105=1075.995,239.417,-82.552,174.560,26.789,154.686
C05106=1075.989,239.169,-82.525,174.557,26.785,154.686
C05107=1075.982,238.920,-82.498,174.555,26.781,154.685
C05108=1075.977,238.671,-82.471,174.553,26.778,154.685
C05109=1075.971,238.423,-82.445,174.551,26.774,154.684
C05110=1075.965,238.175,-82.418,174.548,26.771,154.684
C05111=1075.959,237.926,-82.391,174.546,26.767,154.683
C05112=1075.953,237.678,-82.365,174.543,26.763,154.682
C05113=1075.948,237.430,-82.338,174.541,26.759,154.682
C05114=1075.942,237.181,-82.311,174.539,26.756,154.681
C05115=1075.936,236.932,-82.284,174.536,26.752,154.681
C05116=1075.930,236.683,-82.258,174.534,26.748,154.680
C05117=1075.921,236.276,-82.214,174.530,26.742,154.679
C05118=1075.911,235.869,-82.171,174.527,26.736,154.678
C05119=1075.902,235.462,-82.127,174.523,26.730,154.677
C05120=1075.893,235.054,-82.084,174.518,26.724,154.677
C05121=1075.887,234.805,-82.057,174.516,26.720,154.676
C05122=1075.881,234.557,-82.030,174.514,26.716,154.675
C05123=1075.876,234.309,-82.004,174.512,26.712,154.675
C05124=1075.870,234.060,-81.978,174.509,26.709,154.674
C05125=1075.864,233.811,-81.951,174.507,26.705,154.674
C05126=1075.858,233.563,-81.925,174.505,26.701,154.673
C05127=1075.852,233.314,-81.899,174.503,26.698,154.673
C05128=1075.847,233.066,-81.873,174.500,26.694,154.672
C05129=1075.841,232.818,-81.846,174.498,26.690,154.672
C05130=1075.835,232.569,-81.820,174.495,26.686,154.671
C05131=1075.830,232.320,-81.793,174.493,26.682,154.671
C05132=1075.824,232.072,-81.767,174.491,26.679,154.670
C05133=1075.818,231.823,-81.741,174.488,26.675,154.669
C05134=1075.813,231.575,-81.714,174.486,26.671,154.669
C05135=1075.806,231.326,-81.689,174.484,26.668,154.668
C05136=1075.801,231.078,-81.662,174.482,26.664,154.668
C05137=1075.795,230.829,-81.635,174.479,26.660,154.667
C05138=1075.789,230.580,-81.610,174.477,26.656,154.667
C05139=1075.784,230.332,-81.583,174.475,26.653,154.666
C05140=1075.778,230.083,-81.557,174.473,26.649,154.665
C05141=1075.772,229.835,-81.531,174.470,26.645,154.665
C05142=1075.766,229.586,-81.505,174.467,26.641,154.664
C05143=1075.760,229.338,-81.478,174.465,26.638,154.664
C05144=1075.755,229.089,-81.452,174.463,26.634,154.663
C05145=1075.748,228.841,-81.426,174.461,26.630,154.663
C05146=1075.743,228.592,-81.400,174.459,26.626,154.662
C05147=1075.738,228.343,-81.374,174.456,26.623,154.662
C05148=1075.731,228.094,-81.348,174.454,26.619,154.661
C05149=1075.726,227.846,-81.323,174.452,26.616,154.661
C05150=1075.720,227.597,-81.296,174.450,26.612,154.660
C05151=1075.714,227.348,-81.271,174.447,26.608,154.660
C05152=1075.708,227.099,-81.245,174.445,26.604,154.659
C05153=1075.703,226.852,-81.218,174.443,26.601,154.658
C05154=1075.697,226.603,-81.193,174.441,26.597,154.658
C05155=1075.691,226.354,-81.167,174.439,26.593,154.657
C05156=1075.685,226.106,-81.141,174.435,26.589,154.657
C05157=1075.679,225.857,-81.115,174.433,26.586,154.656
C05158=1075.674,225.608,-81.089,174.431,26.582,154.656
C05159=1075.667,225.360,-81.063,174.429,26.578,154.655
C05160=1075.662,225.111,-81.037,174.426,26.574,154.655
C05161=1075.656,224.862,-81.011,174.424,26.571,154.654
C05162=1075.650,224.614,-80.986,174.422,26.567,154.654
C05163=1075.645,224.366,-80.960,174.420,26.563,154.653
C05164=1075.639,224.117,-80.934,174.418,26.559,154.652
C05165=1075.633,223.868,-80.908,174.415,26.556,154.652
C05166=1075.628,223.619,-80.882,174.413,26.552,154.651
C05167=1075.622,223.371,-80.857,174.411,26.548,154.651
C05168=1075.616,223.122,-80.830,174.409,26.544,154.650
C05169=1075.607,222.707,-80.787,174.405,26.538,154.649
C05170=1075.597,222.291,-80.745,174.402,26.532,154.648
C05171=1075.588,221.876,-80.702,174.398,26.525,154.647
C05172=1075.578,221.459,-80.659,174.394,26.520,154.647
C05173=1075.572,221.211,-80.634,174.392,26.516,154.646
C05174=1075.566,220.963,-80.609,174.390,26.512,154.645
C05175=1075.561,220.714,-80.583,174.388,26.508,154.645
C05176=1075.555,220.465,-80.557,174.385,26.505,154.644
C05177=1075.549,220.216,-80.531,174.383,26.501,154.644
C05178=1075.543,219.968,-80.506,174.381,26.497,154.643
C05179=1075.537,219.720,-80.481,174.379,26.493,154.643
C05180=1075.532,219.471,-80.455,174.376,26.490,154.642
C05181=1075.526,219.222,-80.430,174.374,26.486,154.642
C05182=1075.519,218.973,-80.404,174.371,26.482,154.641
C05183=1075.514,218.724,-80.379,174.369,26.478,154.641
C05184=1075.508,218.476,-80.354,174.367,26.475,154.640
C05185=1075.502,218.228,-80.328,174.364,26.471,154.639
C05186=1075.497,217.979,-80.302,174.362,26.467,154.639
C05187=1075.490,217.730,-80.277,174.360,26.463,154.638
C05188=1075.485,217.482,-80.252,174.358,26.460,154.638
C05189=1075.479,217.233,-80.226,174.356,26.456,154.637
C05190=1075.473,216.984,-80.201,174.353,26.452,154.637
C05191=1075.468,216.736,-80.176,174.351,26.448,154.636
C05192=1075.462,216.487,-80.151,174.349,26.445,154.636
C05193=1075.456,216.238,-80.125,174.348,26.441,154.635
C05194=1075.450,215.989,-80.100,174.346,26.437,154.634
C05195=1075.445,215.741,-80.074,174.344,26.434,154.634
C05196=1075.439,215.492,-80.050,174.341,26.430,154.633
C05197=1075.433,215.243,-80.024,174.339,26.427,154.633
C05198=1075.427,214.995,-79.999,174.337,26.422,154.632
C05199=1075.422,214.746,-79.973,174.335,26.419,154.632
C05200=1075.416,214.497,-79.949,174.333,26.415,154.631
C05201=1075.410,214.249,-79.924,174.330,26.411,154.631
C05202=1075.405,214.000,-79.898,174.328,26.407,154.630
C05203=1075.399,213.751,-79.873,174.326,26.404,154.630
C05204=1075.393,213.503,-79.848,174.324,26.400,154.629
C05205=1075.387,213.254,-79.823,174.322,26.396,154.628
C05206=1075.382,213.006,-79.797,174.319,26.392,154.628
C05207=1075.376,212.757,-79.773,174.317,26.388,154.627
C05208=1075.370,212.508,-79.747,174.315,26.385,154.627
C05209=1075.365,212.260,-79.722,174.313,26.381,154.626
C05210=1075.359,212.011,-79.698,174.311,26.378,154.626
C05211=1075.353,211.762,-79.673,174.309,26.373,154.625
C05212=1075.347,211.513,-79.648,174.306,26.370,154.624
C05213=1075.342,211.264,-79.622,174.304,26.366,154.624
C05214=1075.336,211.016,-79.597,174.302,26.363,154.623
C05215=1075.330,210.767,-79.573,174.300,26.358,154.623
C05216=1075.324,210.518,-79.547,174.298,26.355,154.622
C05217=1075.319,210.270,-79.523,174.295,26.351,154.622
C05218=1075.313,210.021,-79.498,174.293,26.347,154.621
C05219=1075.307,209.772,-79.473,174.291,26.343,154.621
C05220=1075.301,209.524,-79.448,174.289,26.340,154.620
C05221=1075.291,209.112,-79.407,174.285,26.333,154.619
C05222=1075.283,208.701,-79.366,174.283,26.327,154.618
C05223=1075.273,208.289,-79.325,174.279,26.322,154.617
C05224=1075.263,207.878,-79.285,174.275,26.315,154.616
C05225=1075.239,206.839,-79.184,174.157,26.253,154.616
C05226=1075.234,206.591,-79.159,174.154,26.250,154.616
C05227=1075.228,206.342,-79.135,174.152,26.247,154.616
C05228=1075.222,206.093,-79.110,174.150,26.244,154.615
C05229=1075.216,205.845,-79.087,174.147,26.241,154.615
C05230=1075.211,205.596,-79.063,174.145,26.238,154.615
C05231=1075.206,205.347,-79.039,174.143,26.236,154.614
C05232=1075.199,205.098,-79.015,174.141,26.233,154.614
C05233=1075.194,204.849,-78.991,174.139,26.230,154.613
C05234=1075.189,204.601,-78.966,174.136,26.227,154.613
C05235=1075.183,204.352,-78.942,174.134,26.224,154.613
C05236=1075.177,204.103,-78.918,174.132,26.222,154.613
C05237=1075.172,203.854,-78.895,174.129,26.219,154.612
C05238=1075.167,203.605,-78.870,174.127,26.216,154.612
C05239=1075.160,203.357,-78.847,174.125,26.213,154.611
C05240=1075.155,203.109,-78.822,174.123,26.211,154.611
C05241=1075.150,202.859,-78.799,174.121,26.208,154.611
C05242=1075.144,202.610,-78.775,174.118,26.205,154.611
C05243=1075.138,202.362,-78.751,174.116,26.202,154.610
C05244=1075.132,202.114,-78.727,174.113,26.199,154.610
C05245=1075.127,201.864,-78.703,174.111,26.196,154.610
C05246=1075.121,201.615,-78.679,174.109,26.194,154.609
C05247=1075.115,201.367,-78.655,174.107,26.191,154.609
C05248=1075.110,201.118,-78.632,174.105,26.188,154.609
C05249=1075.104,200.869,-78.608,174.102,26.186,154.608
C05250=1075.098,200.620,-78.584,174.100,26.183,154.608
C05251=1075.092,200.371,-78.561,174.098,26.180,154.608
C05252=1075.087,200.123,-78.537,174.095,26.178,154.607
C05253=1075.080,199.873,-78.513,174.093,26.175,154.607
C05254=1075.075,199.625,-78.489,174.091,26.172,154.607
C05255=1075.069,199.376,-78.465,174.089,26.169,154.606
C05256=1075.063,199.127,-78.443,174.087,26.167,154.606
C05257=1075.058,198.879,-78.418,174.084,26.164,154.606
C05258=1075.052,198.629,-78.395,174.082,26.161,154.605
C05259=1075.046,198.381,-78.371,174.079,26.158,154.605
C05260=1075.041,198.132,-78.348,174.078,26.156,154.605
C05261=1075.034,197.884,-78.324,174.076,26.153,154.604
C05262=1075.030,197.634,-78.301,174.073,26.151,154.604
C05263=1075.023,197.386,-78.277,174.071,26.147,154.604
C05264=1075.018,197.136,-78.253,174.069,26.145,154.604
C05265=1075.012,196.888,-78.229,174.066,26.142,154.603
C05266=1075.006,196.639,-78.206,174.065,26.140,154.603
C05267=1075.001,196.390,-78.182,174.062,26.137,154.603
C05268=1074.995,196.141,-78.159,174.060,26.134,154.602
C05269=1074.989,195.893,-78.136,174.058,26.131,154.602
C05270=1074.984,195.644,-78.112,174.055,26.128,154.602
C05271=1074.978,195.395,-78.089,174.054,26.126,154.601
C05272=1074.972,195.146,-78.064,174.051,26.123,154.601
C05273=1074.967,194.897,-78.041,174.049,26.120,154.601
C05274=1074.961,194.649,-78.018,174.047,26.118,154.600
C05275=1074.956,194.399,-77.994,174.044,26.115,154.600
C05276=1074.950,194.151,-77.971,174.043,26.112,154.600
C05277=1074.944,193.902,-77.948,174.040,26.109,154.599
C05278=1074.939,193.653,-77.924,174.038,26.107,154.599
C05279=1074.933,193.404,-77.901,174.036,26.104,154.599
C05280=1074.927,193.156,-77.878,174.033,26.101,154.598
C05281=1074.921,192.907,-77.855,174.032,26.099,154.598
C05282=1074.916,192.658,-77.831,174.029,26.096,154.598
C05283=1074.911,192.409,-77.808,174.027,26.093,154.597
C05284=1074.905,192.161,-77.784,174.025,26.091,154.597
C05285=1074.900,191.911,-77.761,174.023,26.088,154.597
C05286=1074.893,191.630,-77.735,174.020,26.084,154.596
C05287=1074.887,191.349,-77.708,174.018,26.081,154.596
C05288=1074.880,191.068,-77.682,174.015,26.078,154.596
C05289=1074.874,190.788,-77.656,174.013,26.075,154.595
C05290=1074.869,190.538,-77.632,174.011,26.072,154.595
C05291=1074.863,190.289,-77.609,174.009,26.070,154.595
C05292=1074.857,190.041,-77.586,174.007,26.067,154.594
C05293=1074.852,189.791,-77.563,174.004,26.064,154.594
C05294=1074.846,189.543,-77.539,174.002,26.061,154.594
C05295=1074.840,189.294,-77.516,174.001,26.059,154.593
C05296=1074.835,189.045,-77.493,173.998,26.056,154.593
C05297=1074.830,188.796,-77.470,173.996,26.053,154.593
C05298=1074.824,188.547,-77.447,173.993,26.051,154.592
C05299=1074.819,188.299,-77.424,173.992,26.048,154.592
C05300=1074.813,188.050,-77.401,173.990,26.045,154.592
C05301=1074.808,187.801,-77.378,173.987,26.042,154.591
C05302=1074.802,187.552,-77.355,173.985,26.040,154.591
C05303=1074.796,187.304,-77.331,173.984,26.037,154.591
C05304=1074.791,187.055,-77.308,173.981,26.034,154.590
C05305=1074.786,186.806,-77.285,173.979,26.031,154.590
C05306=1074.780,186.557,-77.262,173.976,26.029,154.590
C05307=1074.774,186.308,-77.239,173.975,26.026,154.589
C05308=1074.768,186.059,-77.216,173.973,26.023,154.589
C05309=1074.763,185.811,-77.193,173.970,26.021,154.589
C05310=1074.758,185.562,-77.170,173.969,26.018,154.588
C05311=1074.752,185.313,-77.147,173.966,26.015,154.588
C05312=1074.747,185.063,-77.125,173.964,26.012,154.588
C05313=1074.741,184.814,-77.102,173.962,26.010,154.588
C05314=1074.736,184.565,-77.079,173.960,26.007,154.587
C05315=1074.730,184.316,-77.056,173.958,26.004,154.587
C05316=1074.724,184.068,-77.033,173.956,26.002,154.587
C05317=1074.718,183.819,-77.010,173.953,25.999,154.586
C05318=1074.712,183.570,-76.987,173.952,25.997,154.586
C05319=1074.706,183.321,-76.965,173.949,25.994,154.586
C05320=1074.700,183.072,-76.942,173.947,25.991,154.585
C05321=1074.695,182.823,-76.919,173.945,25.989,154.585
C05322=1074.689,182.574,-76.896,173.943,25.986,154.585
C05323=1074.683,182.325,-76.874,173.941,25.984,154.585
C05324=1074.677,182.076,-76.851,173.939,25.981,154.584
C05325=1074.671,181.827,-76.828,173.937,25.978,154.584
C05326=1074.666,181.579,-76.806,173.934,25.976,154.584
C05327=1074.661,181.330,-76.783,173.932,25.973,154.583
C05328=1074.654,181.081,-76.761,173.931,25.970,154.583
C05329=1074.649,180.832,-76.738,173.928,25.968,154.583
C05330=1074.643,180.583,-76.715,173.926,25.965,154.582
C05331=1074.637,180.334,-76.693,173.924,25.963,154.582
C05332=1074.631,180.085,-76.671,173.922,25.960,154.582
C05333=1074.625,179.836,-76.648,173.920,25.957,154.581
C05334=1074.620,179.587,-76.625,173.918,25.955,154.581
C05335=1074.614,179.338,-76.602,173.916,25.952,154.581
C05336=1074.608,179.090,-76.580,173.913,25.950,154.581
C05337=1074.603,178.841,-76.557,173.912,25.947,154.580
C05338=1074.597,178.592,-76.535,173.909,25.944,154.580
C05339=1074.591,178.343,-76.512,173.907,25.942,154.580
C05340=1074.585,178.094,-76.490,173.906,25.939,154.579
C05341=1074.579,177.845,-76.468,173.903,25.937,154.579
C05342=1074.574,177.596,-76.445,173.901,25.934,154.579
C05343=1074.569,177.348,-76.422,173.899,25.932,154.578
C05344=1074.562,177.098,-76.401,173.897,25.929,154.578
C05345=1074.557,176.849,-76.378,173.895,25.926,154.578
C05346=1074.551,176.600,-76.355,173.893,25.924,154.578
C05347=1074.545,176.351,-76.333,173.891,25.921,154.577
C05348=1074.540,176.103,-76.311,173.888,25.918,154.577
C05349=1074.534,175.854,-76.288,173.887,25.916,154.577
C05350=1074.528,175.573,-76.263,173.885,25.913,154.576
C05351=1074.521,175.291,-76.238,173.882,25.910,154.576
C05352=1074.515,175.010,-76.212,173.880,25.907,154.576
C05353=1074.508,174.728,-76.187,173.878,25.904,154.575
C05354=1074.503,174.480,-76.165,173.875,25.901,154.575
C05355=1074.497,174.230,-76.142,173.874,25.899,154.575
C05356=1074.491,173.981,-76.121,173.872,25.896,154.574
C05357=1074.486,173.733,-76.098,173.869,25.893,154.574
C05358=1074.481,173.483,-76.076,173.868,25.891,154.574
C05359=1074.474,173.235,-76.054,173.865,25.888,154.573
C05360=1074.469,172.985,-76.031,173.863,25.885,154.573
C05361=1074.464,172.737,-76.009,173.861,25.883,154.573
C05362=1074.457,172.488,-75.987,173.859,25.880,154.572
C05363=1074.452,172.239,-75.964,173.858,25.877,154.572
C05364=1074.446,171.989,-75.942,173.855,25.875,154.572
C05365=1074.441,171.741,-75.921,173.853,25.872,154.571
C05366=1074.435,171.492,-75.898,173.852,25.870,154.571
C05367=1074.430,171.243,-75.876,173.849,25.867,154.571
C05368=1074.424,170.994,-75.854,173.847,25.864,154.571
C05369=1074.418,170.745,-75.831,173.845,25.862,154.570
C05370=1074.412,170.496,-75.810,173.843,25.859,154.570
C05371=1074.407,170.248,-75.787,173.842,25.856,154.570
C05372=1074.402,169.998,-75.765,173.839,25.854,154.569
C05373=1074.395,169.749,-75.743,173.837,25.851,154.569
C05374=1074.391,169.500,-75.721,173.835,25.848,154.569
C05375=1074.385,169.251,-75.698,173.833,25.846,154.568
C05376=1074.379,169.003,-75.677,173.832,25.843,154.568
C05377=1074.374,168.753,-75.655,173.829,25.840,154.568
C05378=1074.367,168.505,-75.633,173.828,25.838,154.567
C05379=1074.363,168.256,-75.611,173.825,25.835,154.567
C05380=1074.357,168.006,-75.589,173.823,25.832,154.567
C05381=1074.352,167.758,-75.567,173.822,25.830,154.566
C05382=1074.346,167.508,-75.545,173.819,25.827,154.566
C05383=1074.340,167.260,-75.523,173.818,25.824,154.566
C05384=1074.335,167.011,-75.501,173.815,25.822,154.566
C05385=1074.329,166.761,-75.479,173.813,25.819,154.565
C05386=1074.324,166.513,-75.457,173.812,25.816,154.565
C05387=1074.318,166.263,-75.435,173.809,25.814,154.565
C05388=1074.312,166.015,-75.413,173.808,25.811,154.564
C05389=1074.307,165.766,-75.391,173.806,25.808,154.564
C05390=1074.301,165.517,-75.369,173.804,25.806,154.564
C05391=1074.296,165.268,-75.347,173.802,25.803,154.563
C05392=1074.291,165.018,-75.325,173.799,25.800,154.563
C05393=1074.285,164.770,-75.304,173.798,25.798,154.563
C05394=1074.280,164.520,-75.282,173.796,25.795,154.562
C05395=1074.274,164.272,-75.260,173.794,25.793,154.562
C05396=1074.268,164.023,-75.237,173.792,25.790,154.562
C05397=1074.263,163.775,-75.216,173.790,25.787,154.561
C05398=1074.258,163.525,-75.194,173.788,25.784,154.561
C05399=1074.252,163.277,-75.173,173.787,25.782,154.561
C05400=1074.247,163.027,-75.150,173.784,25.779,154.560
C05401=1074.241,162.778,-75.129,173.783,25.776,154.560
C05402=1074.236,162.529,-75.107,173.781,25.774,154.560
C05403=1074.230,162.280,-75.086,173.778,25.771,154.559
C05404=1074.225,162.031,-75.063,173.777,25.768,154.559
C05405=1074.219,161.782,-75.042,173.774,25.765,154.559
C05406=1074.214,161.533,-75.020,173.773,25.763,154.558
C05407=1074.208,161.284,-74.999,173.771,25.760,154.558
C05408=1074.203,161.035,-74.976,173.769,25.758,154.558
C05409=1074.197,160.786,-74.955,173.767,25.755,154.557
C05410=1074.191,160.537,-74.934,173.765,25.753,154.557
C05411=1074.186,160.288,-74.913,173.763,25.750,154.557
C05412=1074.180,160.039,-74.891,173.762,25.747,154.556
C05413=1074.175,159.790,-74.869,173.759,25.745,154.556
C05414=1074.167,159.508,-74.845,173.757,25.742,154.556
C05415=1074.161,159.227,-74.820,173.755,25.739,154.556
C05416=1074.155,158.945,-74.796,173.753,25.736,154.555
C05417=1074.148,158.664,-74.772,173.751,25.733,154.555
C05418=1074.143,158.414,-74.750,173.749,25.730,154.555
C05419=1074.138,158.165,-74.729,173.747,25.728,154.554
C05420=1074.131,157.916,-74.708,173.745,25.725,154.554
C05421=1074.126,157.668,-74.687,173.743,25.723,154.554
C05422=1074.120,157.418,-74.665,173.741,25.720,154.553
C05423=1074.115,157.169,-74.643,173.740,25.717,154.553
C05424=1074.109,156.920,-74.622,173.737,25.715,154.553
C05425=1074.103,156.671,-74.601,173.736,25.712,154.552
C05426=1074.097,156.422,-74.579,173.733,25.709,154.552
C05427=1074.092,156.173,-74.558,173.732,25.707,154.552
C05428=1074.086,155.924,-74.537,173.730,25.704,154.551
C05429=1074.081,155.675,-74.515,173.728,25.702,154.551
C05430=1074.075,155.426,-74.494,173.726,25.699,154.551
C05431=1074.069,155.177,-74.472,173.724,25.697,154.550
C05432=1074.064,154.928,-74.452,173.722,25.694,154.550
C05433=1074.058,154.679,-74.430,173.721,25.691,154.550
C05434=1074.052,154.430,-74.409,173.718,25.689,154.550
C05435=1074.047,154.180,-74.388,173.717,25.686,154.549
C05436=1074.041,153.932,-74.367,173.714,25.684,154.549
C05437=1074.035,153.683,-74.345,173.713,25.681,154.549
C05438=1074.030,153.434,-74.324,173.711,25.678,154.548
C05439=1074.024,153.185,-74.303,173.709,25.676,154.548
C05440=1074.018,152.936,-74.282,173.707,25.673,154.548
C05441=1074.013,152.687,-74.261,173.706,25.670,154.547
C05442=1074.006,152.438,-74.239,173.703,25.668,154.547
C05443=1074.001,152.189,-74.218,173.702,25.666,154.547
C05444=1073.996,151.940,-74.197,173.699,25.662,154.546
C05445=1073.989,151.691,-74.176,173.698,25.660,154.546
C05446=1073.985,151.441,-74.155,173.696,25.658,154.546
C05447=1073.979,151.192,-74.133,173.694,25.655,154.545
